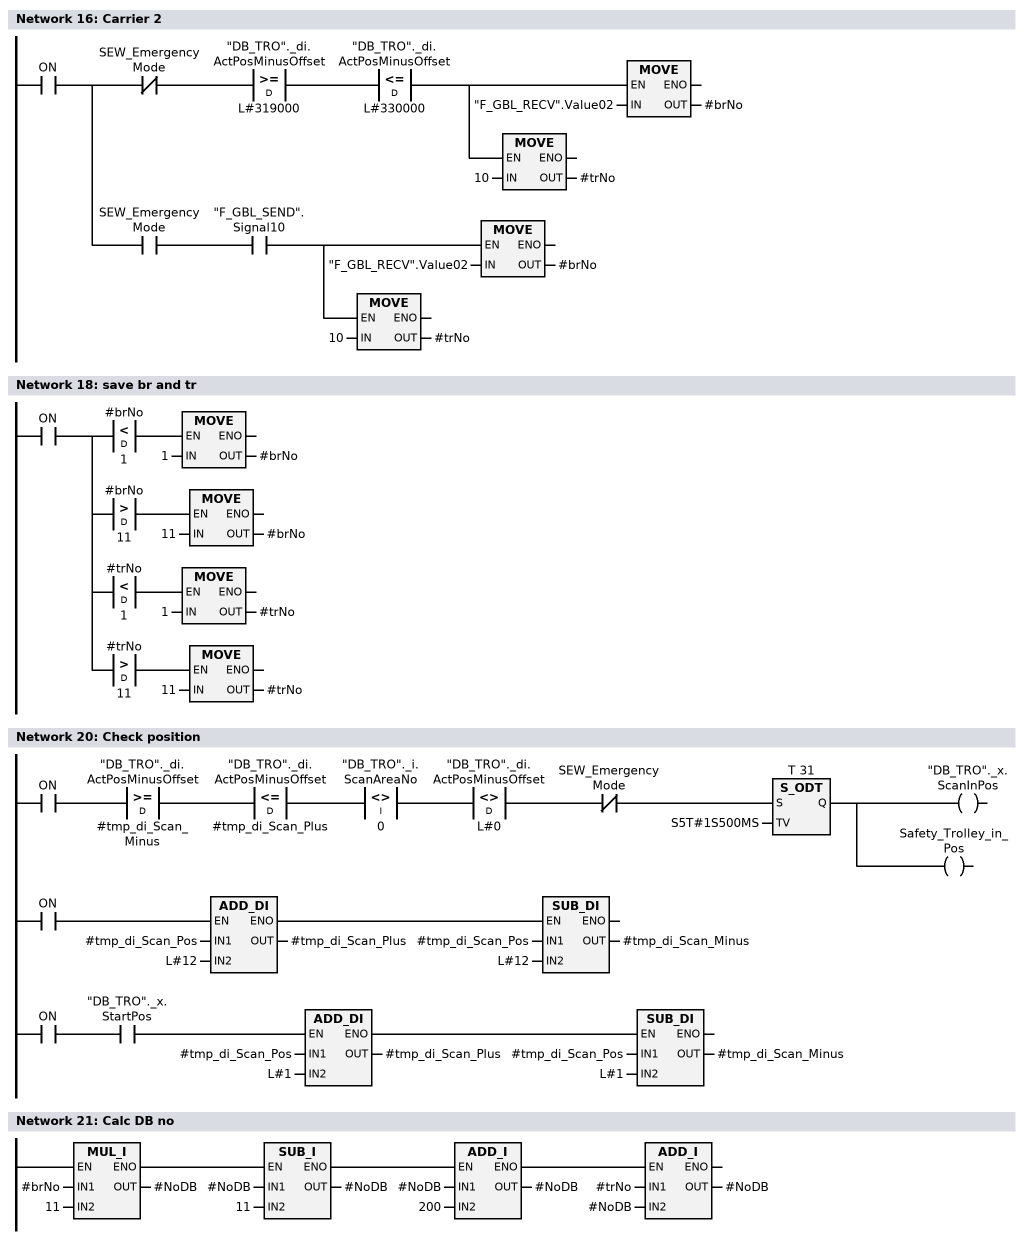
NETWORK
TITLE = Carrier 2
      A     "ON";
      =     L 44.0;
      A     L 44.0;
      AN    "SEW_EmergencyMode";
      A(;
      L     "DB_TRO"._di.ActPosMinusOffset;
      L     L#319000;
      >=D;
      );
      A(;
      L     "DB_TRO"._di.ActPosMinusOffset;
      L     L#330000;
      <=D;
      );
      =     L 44.1;
      A     L 44.1;
      JNB   _01b;
      L     "F_GBL_RECV".Value02;
      T     #brNo;
_01b: NOP   0;
      A     L 44.1;
      JNB   _01c;
      L     10;
      T     #trNo;
_01c: NOP   0;
      A     L 44.0;
      A     "SEW_EmergencyMode";
      A     "F_GBL_SEND".Signal10;
      =     L 44.1;
      A     L 44.1;
      JNB   _01d;
      L     "F_GBL_RECV".Value02;
      T     #brNo;
_01d: NOP   0;
      A     L 44.1;
      JNB   _01e;
      L     10;
      T     #trNo;
_01e: NOP   0;
NETWORK
TITLE = Calc normal row
      L     #trNo;
      L     L#0;
      <>D;
      JC    end;
      L     #startValue;
      L     L#0;
      ==D;
      JC    end;
// we have a row
      L     #brNo;
      L     L#5;
      >D;
      JC    neu;
// old
      L     #startValue;
      L     L#0;	// anpassen auf Achse
      -D;
      DTR;
      L     3.125000e+03;
      /R;
      RND-;
      L     L#2;
      +D;
      T     #trNo;
      JU    end;
// neu
neu:  L     #startValue;
      L     L#0;	// anpassen auf Achse
      -D;
      DTR;
      L     3.500000e+03;
      /R;
      RND-;
      L     L#2;
      +D;
      T     #trNo;
// end
end:  NOP   0;
NETWORK
TITLE = save br and tr
      A     "ON";
      =     L 44.0;
      A     L 44.0;
      A(;
      L     #brNo;
      L     1;
      <D;
      );
      JNB   _01f;
      L     1;
      T     #brNo;
_01f: NOP   0;
      A     L 44.0;
      A(;
      L     #brNo;
      L     11;
      >D;
      );
      JNB   _020;
      L     11;
      T     #brNo;
_020: NOP   0;
      A     L 44.0;
      A(;
      L     #trNo;
      L     1;
      <D;
      );
      JNB   _021;
      L     1;
      T     #trNo;
_021: NOP   0;
      A     L 44.0;
      A(;
      L     #trNo;
      L     11;
      >D;
      );
      JNB   _022;
      L     11;
      T     #trNo;
_022: NOP   0;
NETWORK
TITLE = Get Position
      L     L#0;
      L     "DB_TRO"._i.ScanAreaNo;
      L     1;
      -I;
      L     4;
      *I;
      T     #pMem;
      L     #brNo;
      L     1;
      -I;
      L     44;
      *I;
      L     #pMem;
      +I;
      T     #pMem;
      SLD   3;
      LAR1;
      OPN   "TRO_Positions";
      L     DBD [AR1,P#0.0];
      T     #tmp_di_Scan_Pos;
NETWORK
TITLE = Check position
      A     "ON";
      =     L 44.0;
      A(;
      A     L 44.0;
      JNB   _023;
      L     #tmp_di_Scan_Pos;
      L     L#12;
      +D;
      T     #tmp_di_Scan_Plus;
      AN    OV;
      SAVE;
      CLR;
_023: A     BR;
      );
      JNB   _024;
      L     #tmp_di_Scan_Pos;
      L     L#12;
      -D;
      T     #tmp_di_Scan_Minus;
_024: NOP   0;
      A(;
      A     L 44.0;
      A     "DB_TRO"._x.StartPos;
      JNB   _025;
      L     #tmp_di_Scan_Pos;
      L     L#1;
      +D;
      T     #tmp_di_Scan_Plus;
      AN    OV;
      SAVE;
      CLR;
_025: A     BR;
      );
      JNB   _026;
      L     #tmp_di_Scan_Pos;
      L     L#1;
      -D;
      T     #tmp_di_Scan_Minus;
_026: NOP   0;
      A     L 44.0;
      A(;
      L     "DB_TRO"._di.ActPosMinusOffset;
      L     #tmp_di_Scan_Minus;
      >=D;
      );
      A(;
      L     "DB_TRO"._di.ActPosMinusOffset;
      L     #tmp_di_Scan_Plus;
      <=D;
      );
      A(;
      L     "DB_TRO"._i.ScanAreaNo;
      L     0;
      <>I;
      );
      A(;
      L     "DB_TRO"._di.ActPosMinusOffset;
      L     L#0;
      <>D;
      );
      AN    "SEW_EmergencyMode";
      L     S5T#1S500MS;
      SD    T 31;
      NOP   0;
      NOP   0;
      NOP   0;
      A     T 31;
      =     "DB_TRO"._x.ScanInPos;
      =     "Safety_Trolley_in_Pos";
NETWORK
TITLE = Calc DB no
      A(;
      A(;
      A(;
      L     #brNo;
      L     11;
      *I;
      T     #NoDB;
      AN    OV;
      SAVE;
      CLR;
      A     BR;
      );
      JNB   _027;
      L     #NoDB;
      L     11;
      -I;
      T     #NoDB;
      AN    OV;
      SAVE;
      CLR;
_027: A     BR;
      );
      JNB   _028;
      L     #NoDB;
      L     200;
      +I;
      T     #NoDB;
      AN    OV;
      SAVE;
      CLR;
_028: A     BR;
      );
      JNB   _029;
      L     #trNo;
      L     #NoDB;
      +I;
      T     #NoDB;
_029: NOP   0;
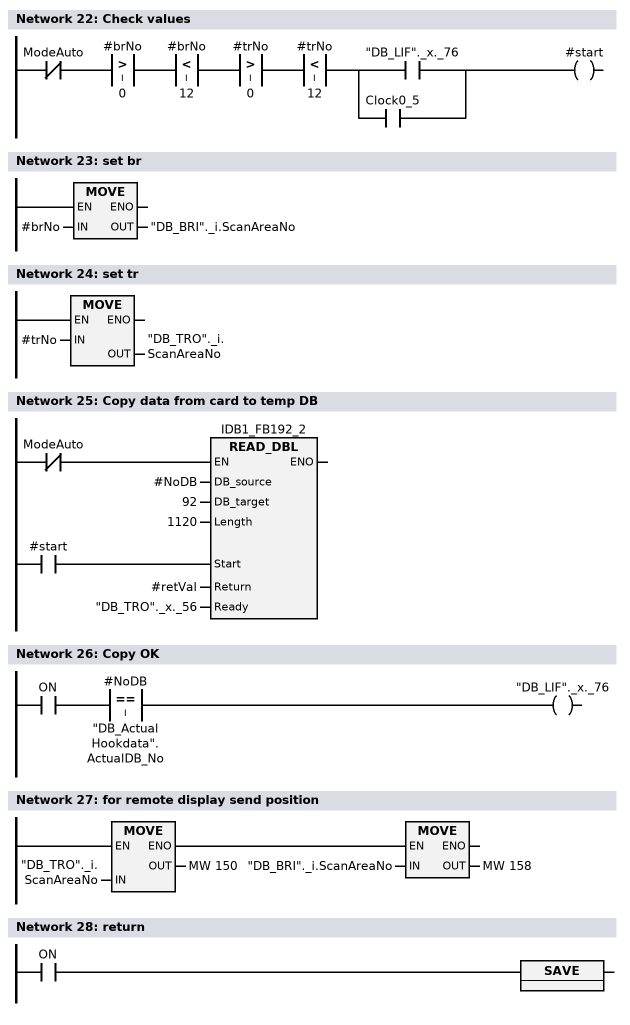
NETWORK
TITLE = Check values
      AN    "ModeAuto";
      A(;
      L     #brNo;
      L     0;
      >I;
      );
      A(;
      L     #brNo;
      L     12;
      <I;
      );
      A(;
      L     #trNo;
      L     0;
      >I;
      );
      A(;
      L     #trNo;
      L     12;
      <I;
      );
      A(;
      O     "DB_LIF"._x._76;
      O     "Clock0_5";
      );
      =     #start;
NETWORK
TITLE = set br
      L     #brNo;
      T     "DB_BRI"._i.ScanAreaNo;
      NOP   0;
NETWORK
TITLE = set tr
      L     #trNo;
      T     "DB_TRO"._i.ScanAreaNo;
      NOP   0;
NETWORK
TITLE = Copy data from card to temp DB
      A     #start;
      =     L 44.0;
      BLD   103;
      AN    "ModeAuto";
      JNB   _02a;
      CALL  "READ_DBL" , "IDB1_FB192_2" (
           DB_source                := #NoDB,
           DB_target                := 92,
           Length                   := 1120,
           Start                    := L 44.0,
           Return                   := #retVal,
           Ready                    := "DB_TRO"._x._56);
_02a: NOP   0;
NETWORK
TITLE = Copy OK
      A     "ON";
      A(;
      L     #NoDB;
      L     "DB_ActualHookdata".ActualDB_No;
      ==I;
      );
      =     "DB_LIF"._x._76;
NETWORK
TITLE = for remote display send position
      A(;
      L     "DB_TRO"._i.ScanAreaNo;
      T     MW 150;
      SET;
      SAVE;
      CLR;
      A     BR;
      );
      JNB   _02b;
      L     "DB_BRI"._i.ScanAreaNo;
      T     MW 158;
_02b: NOP   0;
NETWORK
TITLE = return
      A     "ON";
      SAVE;
END_FUNCTION

FUNCTION "Axis_TROLLEY_Scan_Man" : VOID	// FC 215
TITLE = Scan manual pos
//
//Baustein-Kommentar ...
//
AUTHOR : Koenig
FAMILY : Scan
NAME : ManPos
VERSION : 1.0
VAR_INPUT
  BridgeNo : INT ;	//Bridge position no
  PositionNo : INT ;	//Positions number
  PositionDB : INT ;	//DB Number of Positions
  ActualPosition : DINT ;
  PositionMin : DINT ;
  PositionMax : DINT ;
END_VAR
VAR_OUTPUT
  PrevPosition : DINT ;
  NextPosition : DINT ;
  FirstPosition : DINT ;
  LastPosition : DINT ;
  Error : WORD ;
END_VAR
VAR_TEMP
  i : INT ;
  value : DINT ;
  diff : DINT ;
  DB_No : WORD ;
  DB_Length : WORD ;
  DB_WP : BOOL ;
  RETURN_Value : INT ;
END_VAR
BEGIN
// body was compiled from an SCL source; compiled code not shown
END_FUNCTION

FUNCTION "Axis_TROLLEY_Flt_065-080" : VOID	// FC 219
TITLE = Error Trolley 65-80
VERSION : 0.1
BEGIN
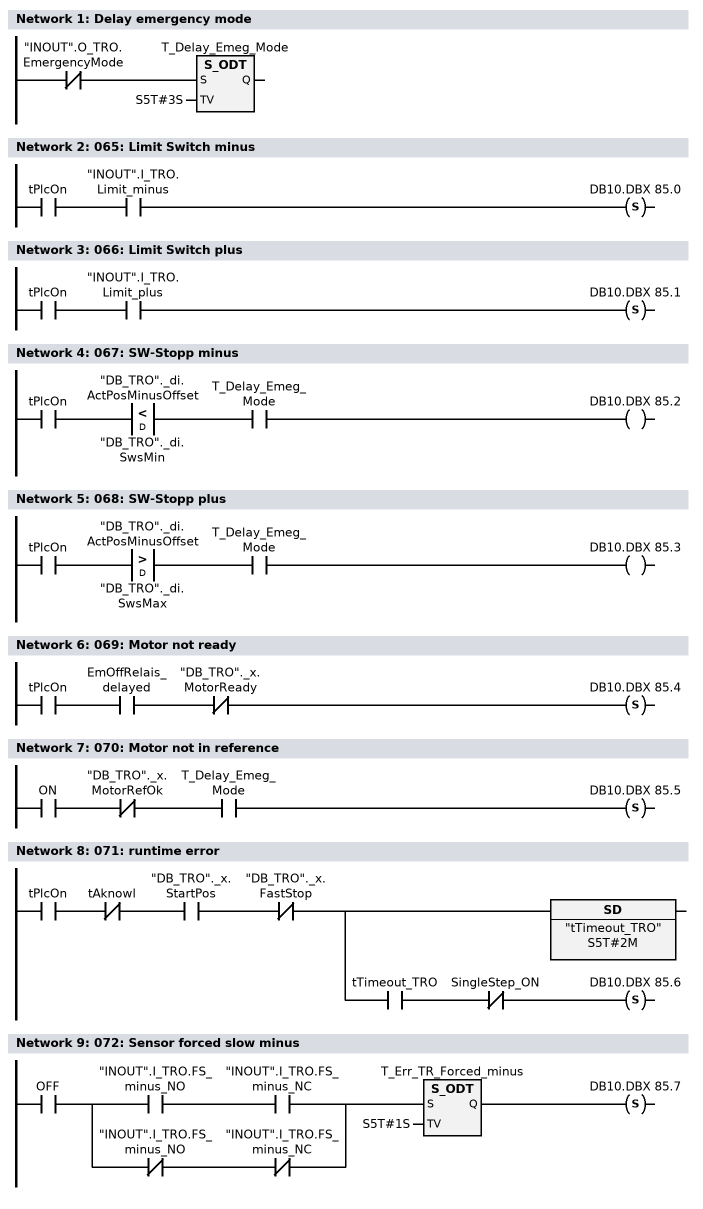
NETWORK
TITLE = Delay emergency mode
      AN    "INOUT".O_TRO.EmergencyMode;
      L     S5T#3S;
      SD    "T_Delay_Emeg_Mode";
      NOP   0;
      NOP   0;
      NOP   0;
      NOP   0;
NETWORK
TITLE = 065: Limit Switch minus
      A     "tPlcOn";
      A     "INOUT".I_TRO.Limit_minus;
      S     DB10.DBX 85.0;
NETWORK
TITLE = 066: Limit Switch plus
      A     "tPlcOn";
      A     "INOUT".I_TRO.Limit_plus;
      S     DB10.DBX 85.1;
NETWORK
TITLE = 067: SW-Stopp minus
      A     "tPlcOn";
      A(;
      L     "DB_TRO"._di.ActPosMinusOffset;
      L     "DB_TRO"._di.SwsMin;
      <D;
      );
      A     "T_Delay_Emeg_Mode";
      =     DB10.DBX 85.2;
NETWORK
TITLE = 068: SW-Stopp plus
      A     "tPlcOn";
      A(;
      L     "DB_TRO"._di.ActPosMinusOffset;
      L     "DB_TRO"._di.SwsMax;
      >D;
      );
      A     "T_Delay_Emeg_Mode";
      =     DB10.DBX 85.3;
NETWORK
TITLE = 069: Motor not ready
      A     "tPlcOn";
      A     "EmOffRelais_delayed";
      AN    "DB_TRO"._x.MotorReady;
      S     DB10.DBX 85.4;
NETWORK
TITLE = 070: Motor not in reference
      A     "ON";
      AN    "DB_TRO"._x.MotorRefOk;
      A     "T_Delay_Emeg_Mode";
      S     DB10.DBX 85.5;
NETWORK
TITLE = 071: runtime error
      A     "tPlcOn";
      AN    "tAknowl";
      A     "DB_TRO"._x.StartPos;
      AN    "DB_TRO"._x.FastStop;
      =     L 0.0;
      A     L 0.0;
      BLD   102;
      L     S5T#2M;
      SD    "tTimeout_TRO";
      A     L 0.0;
      A     "tTimeout_TRO";
      AN    "SingleStep_ON";
      S     DB10.DBX 85.6;
NETWORK
TITLE = 072: Sensor forced slow minus
      A     "OFF";
      A(;
      A     "INOUT".I_TRO.FS_minus_NO;
      A     "INOUT".I_TRO.FS_minus_NC;
      O;
      AN    "INOUT".I_TRO.FS_minus_NO;
      AN    "INOUT".I_TRO.FS_minus_NC;
      );
      L     S5T#1S;
      SD    "T_Err_TR_Forced_minus";
      NOP   0;
      NOP   0;
      NOP   0;
      A     "T_Err_TR_Forced_minus";
      S     DB10.DBX 85.7;
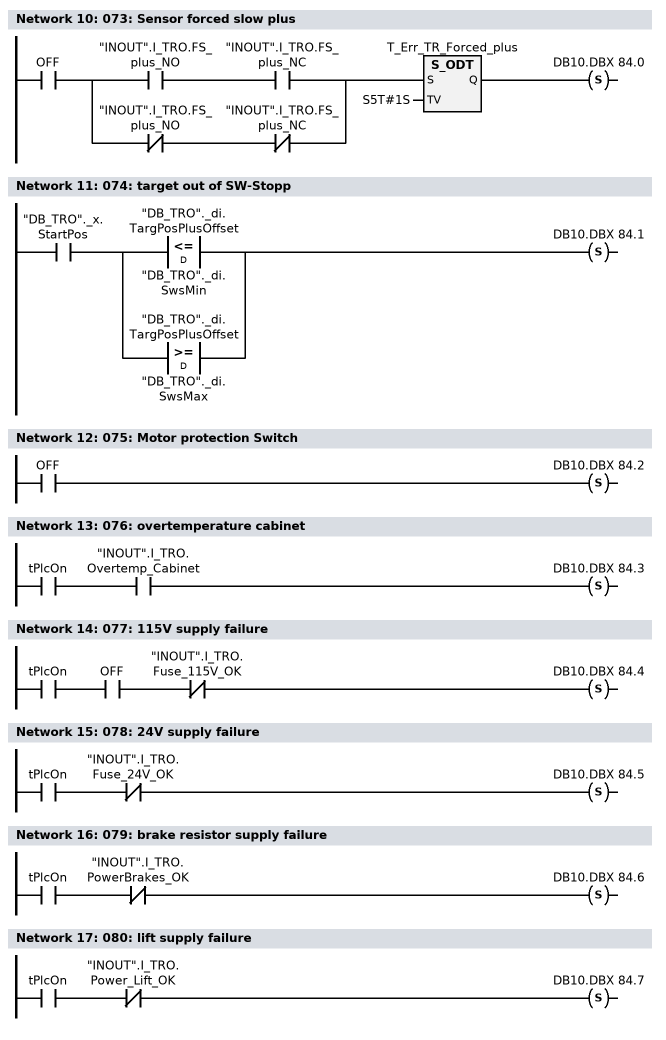
NETWORK
TITLE = 073: Sensor forced slow plus
      A     "OFF";
      A(;
      A     "INOUT".I_TRO.FS_plus_NO;
      A     "INOUT".I_TRO.FS_plus_NC;
      O;
      AN    "INOUT".I_TRO.FS_plus_NO;
      AN    "INOUT".I_TRO.FS_plus_NC;
      );
      L     S5T#1S;
      SD    "T_Err_TR_Forced_plus";
      NOP   0;
      NOP   0;
      NOP   0;
      A     "T_Err_TR_Forced_plus";
      S     DB10.DBX 84.0;
NETWORK
TITLE = 074: target out of SW-Stopp
      A     "DB_TRO"._x.StartPos;
      A(;
      O(;
      L     "DB_TRO"._di.TargPosPlusOffset;
      L     "DB_TRO"._di.SwsMin;
      <=D;
      );
      O(;
      L     "DB_TRO"._di.TargPosPlusOffset;
      L     "DB_TRO"._di.SwsMax;
      >=D;
      );
      );
      S     DB10.DBX 84.1;
NETWORK
TITLE = 075: Motor protection Switch
      A     "OFF";
      S     DB10.DBX 84.2;
NETWORK
TITLE = 076: overtemperature cabinet
      A     "tPlcOn";
      A     "INOUT".I_TRO.Overtemp_Cabinet;
      S     DB10.DBX 84.3;
NETWORK
TITLE = 077: 115V supply failure
      A     "tPlcOn";
      A     "OFF";
      AN    "INOUT".I_TRO.Fuse_115V_OK;
      S     DB10.DBX 84.4;
NETWORK
TITLE = 078: 24V supply failure
      A     "tPlcOn";
      AN    "INOUT".I_TRO.Fuse_24V_OK;
      S     DB10.DBX 84.5;
NETWORK
TITLE = 079: brake resistor supply failure
//14 
      A     "tPlcOn";
      AN    "INOUT".I_TRO.PowerBrakes_OK;
      S     DB10.DBX 84.6;
NETWORK
TITLE = 080: lift supply failure
      A     "tPlcOn";
      AN    "INOUT".I_TRO.Power_Lift_OK;
      S     DB10.DBX 84.7;
END_FUNCTION

FUNCTION "Axis_LIFT" : VOID	// FC 220
TITLE = Axis LIFT
VERSION : 0.1
VAR_TEMP
  tmp_RetVal : INT ;
  tmp_RetVal2 : INT ;
  tmp_SourceDB1 : INT ;
  tmp_SourceDB2 : INT ;
  tmp_TargetDB1 : INT ;
  tmp_TargetDB2 : INT ;
  tmp_StartDBCopy : BOOL ;
  tmp_ReadDB_OK : BOOL ;
END_VAR
BEGIN
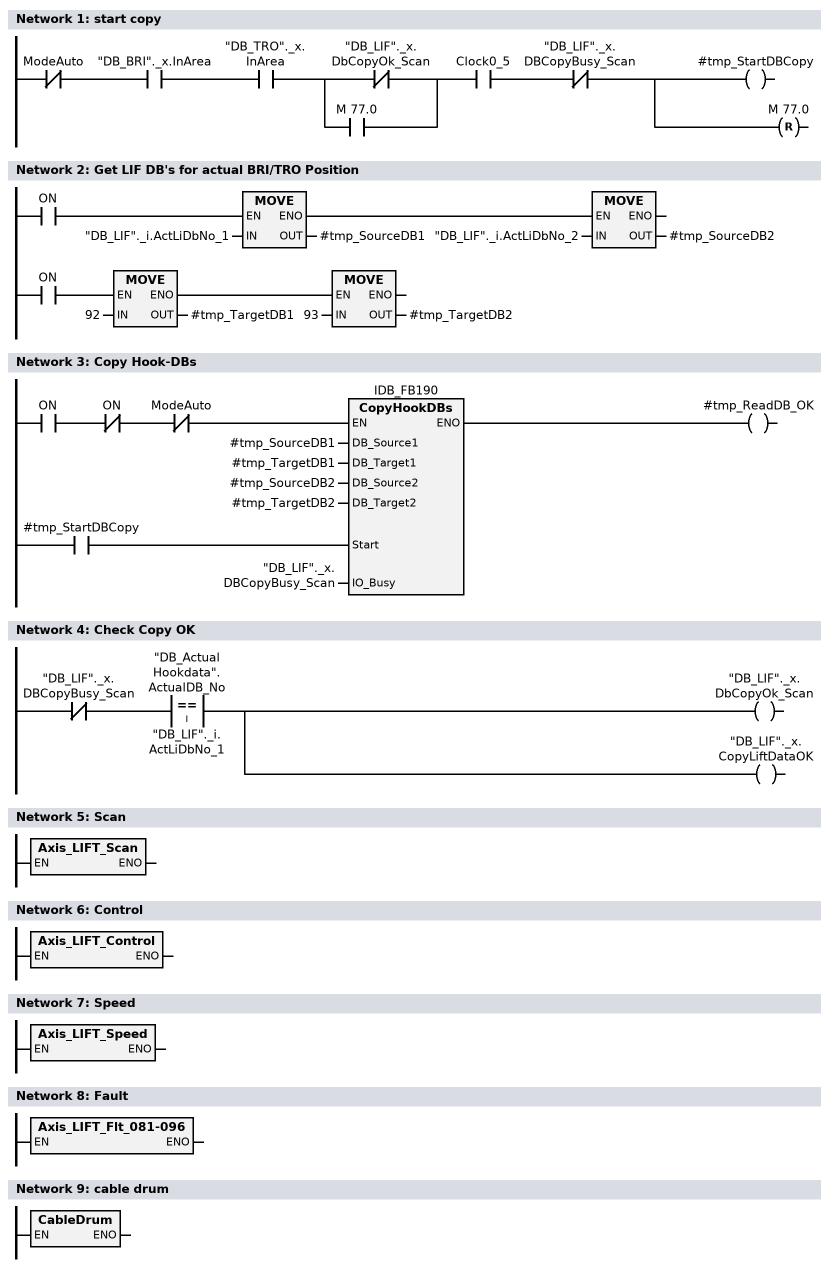
NETWORK
TITLE = start copy
      AN    "ModeAuto";
      A     "DB_BRI"._x.InArea;
      A     "DB_TRO"._x.InArea;
      A(;
      ON    "DB_LIF"._x.DbCopyOk_Scan;
      O     M 77.0;
      );
      A     "Clock0_5";
      AN    "DB_LIF"._x.DBCopyBusy_Scan;
      =     #tmp_StartDBCopy;
      R     M 77.0;
NETWORK
TITLE = Get LIF DB's for actual BRI/TRO Position
//Actual DB from Scan BRI
//
      A     "ON";
      =     L 13.0;
      A(;
      A     L 13.0;
      JNB   _001;
      L     "DB_LIF"._i.ActLiDbNo_1;
      T     #tmp_SourceDB1;
      SET;
      SAVE;
      CLR;
_001: A     BR;
      );
      JNB   _002;
      L     "DB_LIF"._i.ActLiDbNo_2;
      T     #tmp_SourceDB2;
_002: NOP   0;
      A(;
      A     L 13.0;
      JNB   _003;
      L     92;
      T     #tmp_TargetDB1;
      SET;
      SAVE;
      CLR;
_003: A     BR;
      );
      JNB   _004;
      L     93;
      T     #tmp_TargetDB2;
_004: NOP   0;
NETWORK
TITLE = Copy Hook-DBs
      A     #tmp_StartDBCopy;
      =     L 13.0;
      BLD   103;
      A     "ON";
      AN    "ON";
      AN    "ModeAuto";
      JNB   _005;
      CALL  "CopyHookDBs" , "IDB_FB190" (
           DB_Source1               := #tmp_SourceDB1,
           DB_Target1               := #tmp_TargetDB1,
           DB_Source2               := #tmp_SourceDB2,
           DB_Target2               := #tmp_TargetDB2,
           Start                    := L 13.0,
           IO_Busy                  := "DB_LIF"._x.DBCopyBusy_Scan);
_005: A     BR;
      =     #tmp_ReadDB_OK;
NETWORK
TITLE = Check Copy OK
      AN    "DB_LIF"._x.DBCopyBusy_Scan;
      A(;
      L     "DB_ActualHookdata".ActualDB_No;
      L     "DB_LIF"._i.ActLiDbNo_1;
      ==I;
      );
      =     "DB_LIF"._x.DbCopyOk_Scan;
      =     "DB_LIF"._x.CopyLiftDataOK;
NETWORK
TITLE = Scan
      CALL  "Axis_LIFT_Scan";
      NOP   0;
NETWORK
TITLE = Control
      CALL  "Axis_LIFT_Control";
      NOP   0;
NETWORK
TITLE = Speed
      CALL  "Axis_LIFT_Speed";
      NOP   0;
NETWORK
TITLE = Fault
      CALL  "Axis_LIFT_Flt_081-096";
      NOP   0;
NETWORK
TITLE = cable drum
      CALL  "CableDrum";
      NOP   0;
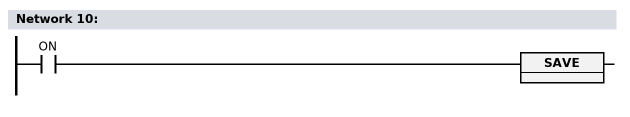
NETWORK
TITLE =
      A     "ON";
      SAVE;
END_FUNCTION

FUNCTION "Axis_LIFT_Control" : VOID	// FC 222
TITLE = LIFT Control
VERSION : 0.1
VAR_TEMP
  tmp_Targ_HO_1_auto : BOOL ;
  tmp_Targ_HO_2_auto : BOOL ;
  tmp_Targ_HO_3_auto : BOOL ;
  tmp_Targ_HO_1_man : BOOL ;
  tmp_Targ_HU_1_auto : BOOL ;
  tmp_Targ_HU_2_auto : BOOL ;
  tmp_Targ_HU_1_man : BOOL ;
  tmp_Targ_Intern_1_auto : BOOL ;
  tmp_Targ_Intern_2_auto : BOOL ;
  tmp_Targ_Intern_3_auto : BOOL ;
  tmp_Targ_Top_auto : BOOL ;
  tmp_Targ_Top_man : BOOL ;
  tmp_switch : BOOL ;
  TargetOK : BOOL ;
  TargetValueOK : BOOL ;
  tmp_InPos : BOOL ;
  tmp_Rel_MaxDis : BOOL ;
  modePos : BOOL ;
  modeInch : BOOL ;
  tmp_Targ_Man : BOOL ;
  tmp_DIR : BOOL ;
  tmp_di_DiffPos : DINT ;
  prev : DINT ;
  next : DINT ;
  min : DINT ;
  max : DINT ;
END_VAR
BEGIN
NETWORK
TITLE =
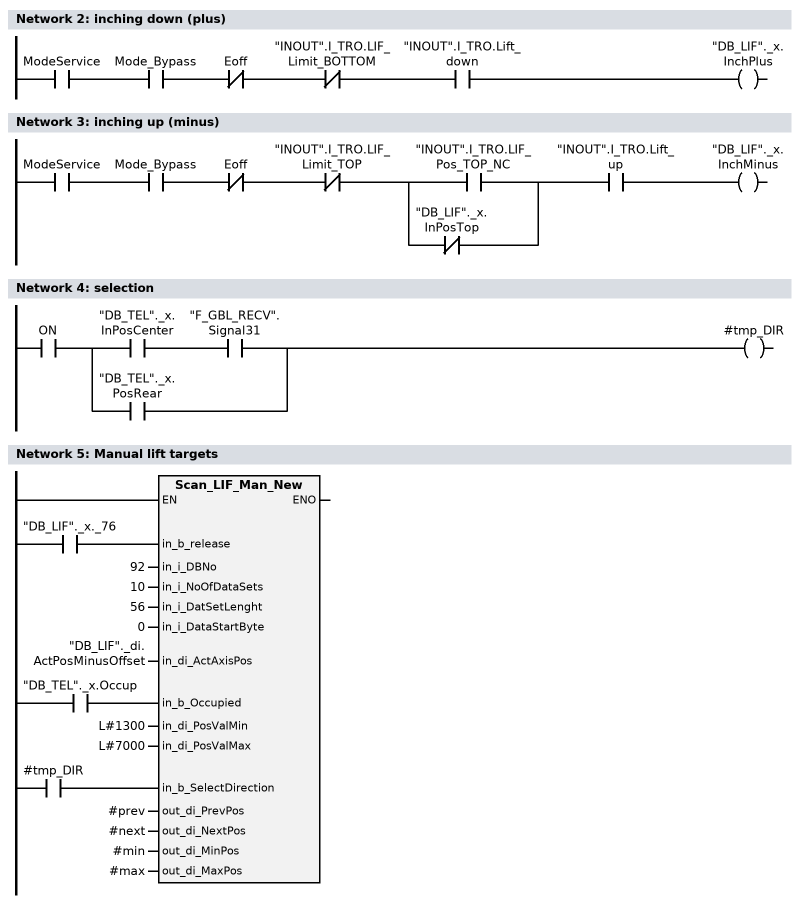
NETWORK
TITLE = inching down (plus)
      A     "ModeService";
      A     "Mode_Bypass";
      AN    "Eoff";
      AN    "INOUT".I_TRO.LIF_Limit_BOTTOM;
      A     "INOUT".I_TRO.Lift_down;
      =     "DB_LIF"._x.InchPlus;
NETWORK
TITLE = inching up (minus)
      A     "ModeService";
      A     "Mode_Bypass";
      AN    "Eoff";
      AN    "INOUT".I_TRO.LIF_Limit_TOP;
      A(;
      O     "INOUT".I_TRO.LIF_Pos_TOP_NC;
      ON    "DB_LIF"._x.InPosTop;
      );
      A     "INOUT".I_TRO.Lift_up;
      =     "DB_LIF"._x.InchMinus;
NETWORK
TITLE = selection
      A     "ON";
      A(;
      A     "DB_TEL"._x.InPosCenter;
      A     "F_GBL_RECV".Signal31;
      O     "DB_TEL"._x.PosRear;
      );
      =     #tmp_DIR;
NETWORK
TITLE = Manual lift targets
      A     "DB_LIF"._x._76;
      =     L 24.0;
      BLD   103;
      A     "DB_TEL"._x.Occup;
      =     L 24.1;
      BLD   103;
      A     #tmp_DIR;
      =     L 24.2;
      BLD   103;
      CALL  "Scan_LIF_Man_New" (
           in_b_release             := L 24.0,
           in_i_DBNo                := 92,
           in_i_NoOfDataSets        := 10,
           in_i_DatSetLenght        := 56,
           in_i_DataStartByte       := 0,
           in_di_ActAxisPos         := "DB_LIF"._di.ActPosMinusOffset,
           in_b_Occupied            := L 24.1,
           in_di_PosValMin          := L#1300,
           in_di_PosValMax          := L#7000,
           in_b_SelectDirection     := L 24.2,
           out_di_PrevPos           := #prev,
           out_di_NextPos           := #next,
           out_di_MinPos            := #min,
           out_di_MaxPos            := #max);
      NOP   0;
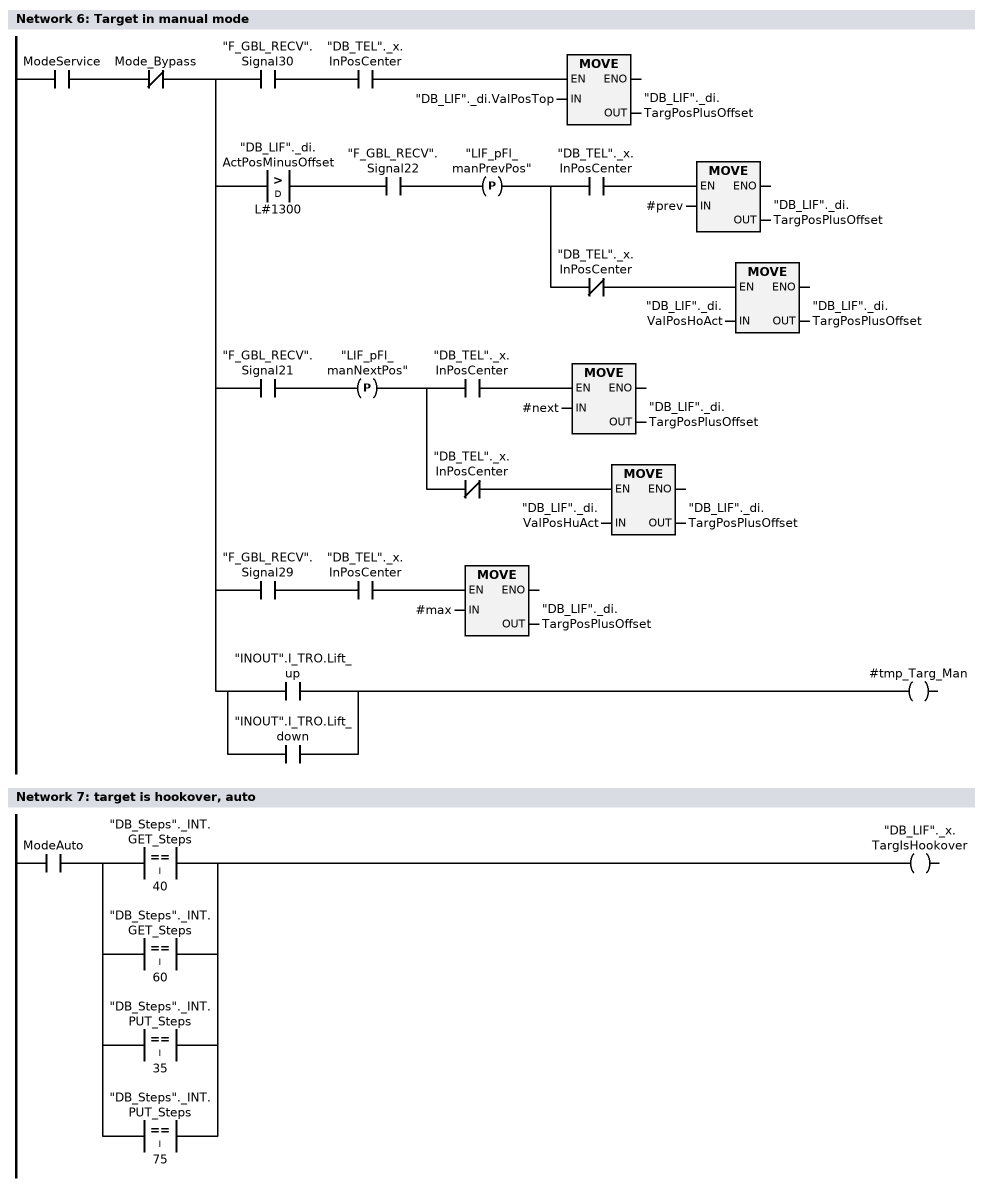
NETWORK
TITLE = Target in manual mode
      A     "ModeService";
      AN    "Mode_Bypass";
      =     L 24.0;
      A     L 24.0;
      A     "F_GBL_RECV".Signal30;
      A     "DB_TEL"._x.InPosCenter;
      JNB   _001;
      L     "DB_LIF"._di.ValPosTop;
      T     "DB_LIF"._di.TargPosPlusOffset;
_001: NOP   0;
      A     L 24.0;
      A(;
      L     "DB_LIF"._di.ActPosMinusOffset;
      L     L#1300;
      >D;
      );
      A     "F_GBL_RECV".Signal22;
      FP    "LIF_pFl_manPrevPos";
      =     L 24.1;
      A     L 24.1;
      A     "DB_TEL"._x.InPosCenter;
      JNB   _002;
      L     #prev;
      T     "DB_LIF"._di.TargPosPlusOffset;
_002: NOP   0;
      A     L 24.1;
      AN    "DB_TEL"._x.InPosCenter;
      JNB   _003;
      L     "DB_LIF"._di.ValPosHoAct;
      T     "DB_LIF"._di.TargPosPlusOffset;
_003: NOP   0;
      A     L 24.0;
      A     "F_GBL_RECV".Signal21;
      FP    "LIF_pFl_manNextPos";
      =     L 24.1;
      A     L 24.1;
      A     "DB_TEL"._x.InPosCenter;
      JNB   _004;
      L     #next;
      T     "DB_LIF"._di.TargPosPlusOffset;
_004: NOP   0;
      A     L 24.1;
      AN    "DB_TEL"._x.InPosCenter;
      JNB   _005;
      L     "DB_LIF"._di.ValPosHuAct;
      T     "DB_LIF"._di.TargPosPlusOffset;
_005: NOP   0;
      A     L 24.0;
      A     "F_GBL_RECV".Signal29;
      A     "DB_TEL"._x.InPosCenter;
      JNB   _006;
      L     #max;
      T     "DB_LIF"._di.TargPosPlusOffset;
_006: NOP   0;
      A     L 24.0;
      A(;
      O     "INOUT".I_TRO.Lift_up;
      O     "INOUT".I_TRO.Lift_down;
      );
      =     #tmp_Targ_Man;
NETWORK
TITLE = target is hookover, auto
      A     "ModeAuto";
      A(;
      O(;
      L     "DB_Steps"._INT.GET_Steps;
      L     40;
      ==I;
      );
      O(;
      L     "DB_Steps"._INT.GET_Steps;
      L     60;
      ==I;
      );
      O(;
      L     "DB_Steps"._INT.PUT_Steps;
      L     35;
      ==I;
      );
      O(;
      L     "DB_Steps"._INT.PUT_Steps;
      L     75;
      ==I;
      );
      );
      =     "DB_LIF"._x.TargIsHookover;
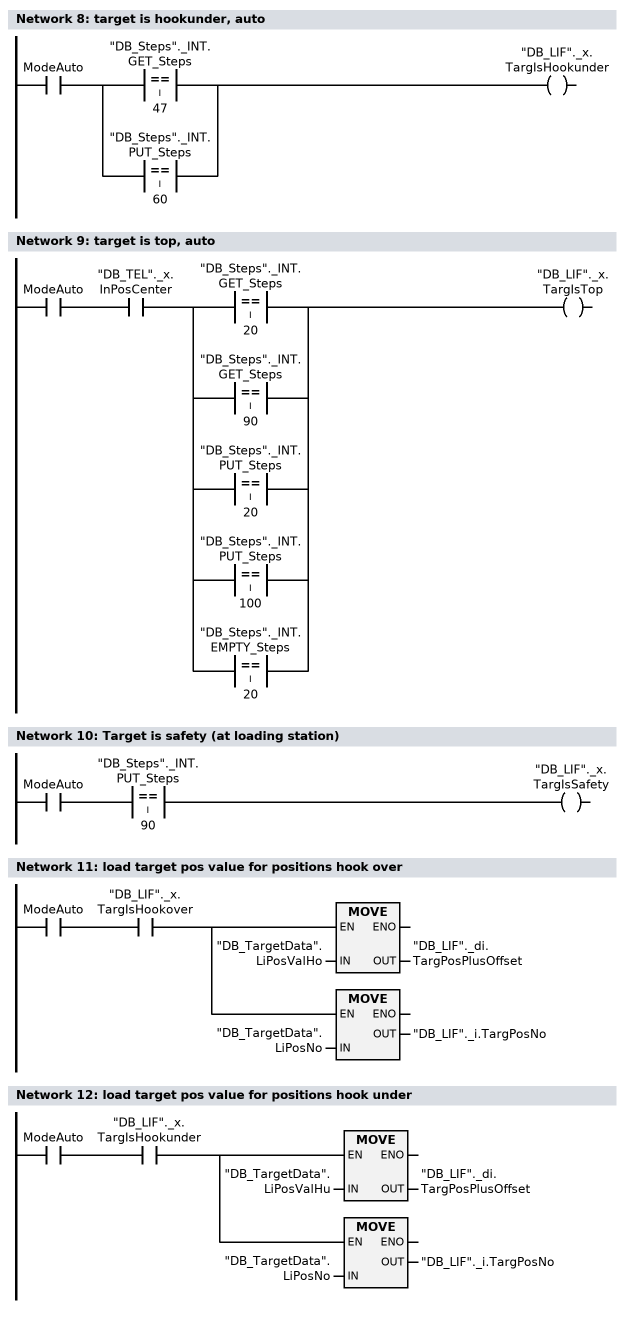
NETWORK
TITLE = target is hookunder, auto
      A     "ModeAuto";
      A(;
      O(;
      L     "DB_Steps"._INT.GET_Steps;
      L     47;
      ==I;
      );
      O(;
      L     "DB_Steps"._INT.PUT_Steps;
      L     60;
      ==I;
      );
      );
      =     "DB_LIF"._x.TargIsHookunder;
NETWORK
TITLE = target is top, auto
      A     "ModeAuto";
      A     "DB_TEL"._x.InPosCenter;
      A(;
      O(;
      L     "DB_Steps"._INT.GET_Steps;
      L     20;
      ==I;
      );
      O(;
      L     "DB_Steps"._INT.GET_Steps;
      L     90;
      ==I;
      );
      O(;
      L     "DB_Steps"._INT.PUT_Steps;
      L     20;
      ==I;
      );
      O(;
      L     "DB_Steps"._INT.PUT_Steps;
      L     100;
      ==I;
      );
      O(;
      L     "DB_Steps"._INT.EMPTY_Steps;
      L     20;
      ==I;
      );
      );
      =     "DB_LIF"._x.TargIsTop;
NETWORK
TITLE = Target is safety (at loading station)
      A     "ModeAuto";
      A(;
      L     "DB_Steps"._INT.PUT_Steps;
      L     90;
      ==I;
      );
      =     "DB_LIF"._x.TargIsSafety;
NETWORK
TITLE = load target pos value for positions hook over
      A     "ModeAuto";
      A     "DB_LIF"._x.TargIsHookover;
      =     L 24.0;
      A     L 24.0;
      JNB   _007;
      L     "DB_TargetData".LiPosValHo;
      T     "DB_LIF"._di.TargPosPlusOffset;
_007: NOP   0;
      A     L 24.0;
      JNB   _008;
      L     "DB_TargetData".LiPosNo;
      T     "DB_LIF"._i.TargPosNo;
_008: NOP   0;
NETWORK
TITLE = load target pos value for positions hook under
      A     "ModeAuto";
      A     "DB_LIF"._x.TargIsHookunder;
      =     L 24.0;
      A     L 24.0;
      JNB   _009;
      L     "DB_TargetData".LiPosValHu;
      T     "DB_LIF"._di.TargPosPlusOffset;
_009: NOP   0;
      A     L 24.0;
      JNB   _00a;
      L     "DB_TargetData".LiPosNo;
      T     "DB_LIF"._i.TargPosNo;
_00a: NOP   0;
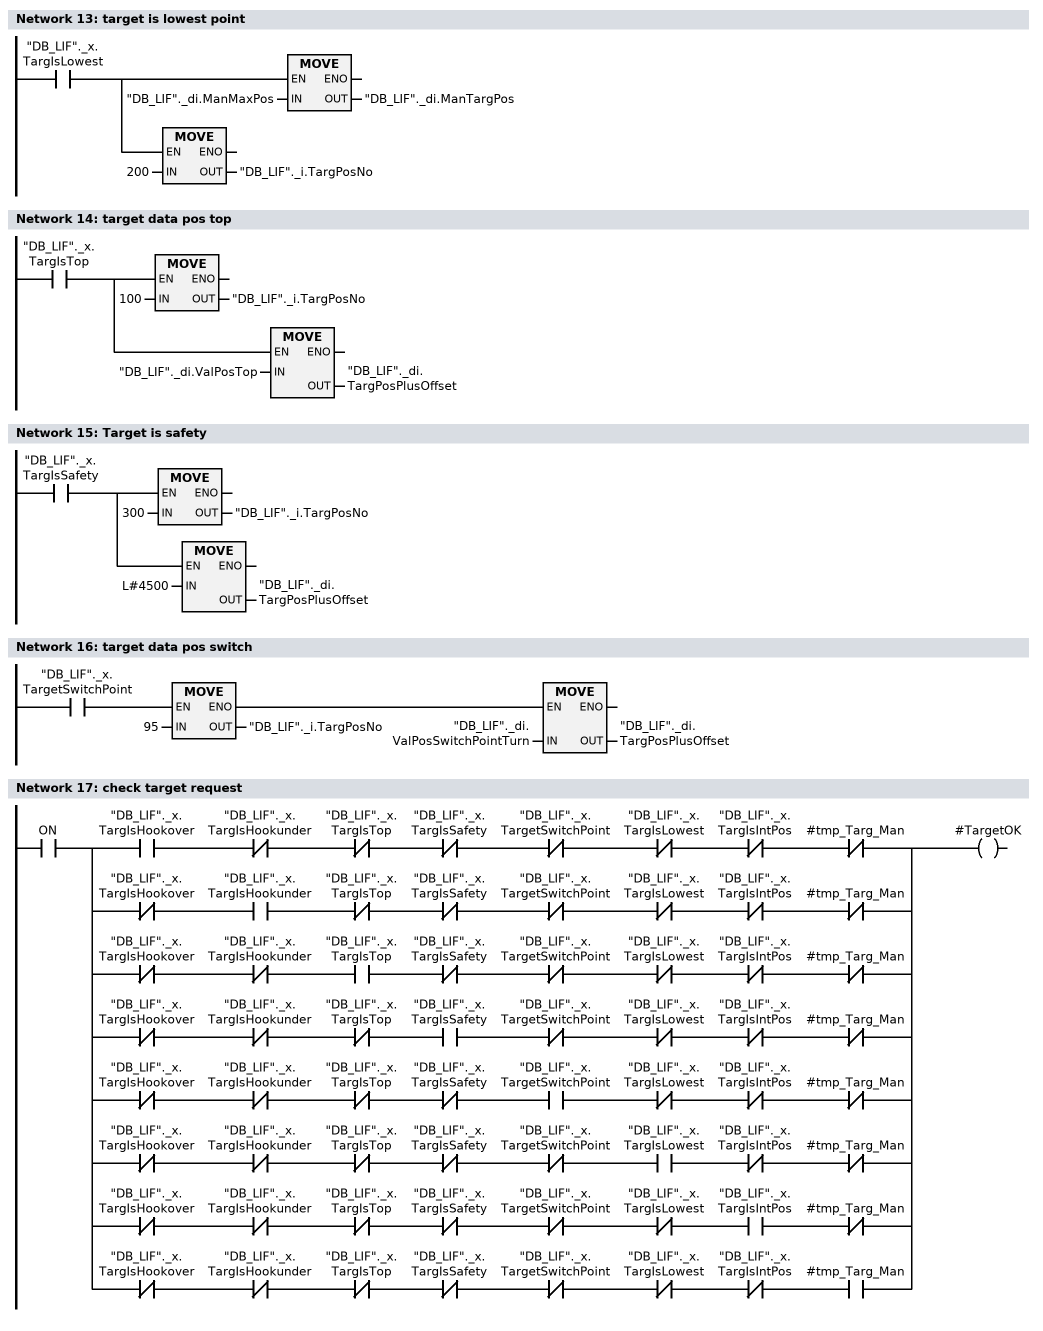
NETWORK
TITLE = target is lowest point
      A     "DB_LIF"._x.TargIsLowest;
      =     L 24.0;
      A     L 24.0;
      JNB   _00b;
      L     "DB_LIF"._di.ManMaxPos;
      T     "DB_LIF"._di.ManTargPos;
_00b: NOP   0;
      A     L 24.0;
      JNB   _00c;
      L     200;
      T     "DB_LIF"._i.TargPosNo;
_00c: NOP   0;
NETWORK
TITLE = target data pos top
      A     "DB_LIF"._x.TargIsTop;
      =     L 24.0;
      A     L 24.0;
      JNB   _00d;
      L     100;
      T     "DB_LIF"._i.TargPosNo;
_00d: NOP   0;
      A     L 24.0;
      JNB   _00e;
      L     "DB_LIF"._di.ValPosTop;
      T     "DB_LIF"._di.TargPosPlusOffset;
_00e: NOP   0;
NETWORK
TITLE = Target is safety
      A     "DB_LIF"._x.TargIsSafety;
      =     L 24.0;
      A     L 24.0;
      JNB   _00f;
      L     300;
      T     "DB_LIF"._i.TargPosNo;
_00f: NOP   0;
      A     L 24.0;
      JNB   _010;
      L     L#4500;
      T     "DB_LIF"._di.TargPosPlusOffset;
_010: NOP   0;
NETWORK
TITLE = target data pos switch
      A(;
      A     "DB_LIF"._x.TargetSwitchPoint;
      JNB   _011;
      L     95;
      T     "DB_LIF"._i.TargPosNo;
      SET;
      SAVE;
      CLR;
_011: A     BR;
      );
      JNB   _012;
      L     "DB_LIF"._di.ValPosSwitchPointTurn;
      T     "DB_LIF"._di.TargPosPlusOffset;
_012: NOP   0;
NETWORK
TITLE = check target request
//only allow one target otherwise values are wrong !
      A     "ON";
      A(;
      A     "DB_LIF"._x.TargIsHookover;
      AN    "DB_LIF"._x.TargIsHookunder;
      AN    "DB_LIF"._x.TargIsTop;
      AN    "DB_LIF"._x.TargIsSafety;
      AN    "DB_LIF"._x.TargetSwitchPoint;
      AN    "DB_LIF"._x.TargIsLowest;
      AN    "DB_LIF"._x.TargIsIntPos;
      AN    #tmp_Targ_Man;
      O;
      AN    "DB_LIF"._x.TargIsHookover;
      A     "DB_LIF"._x.TargIsHookunder;
      AN    "DB_LIF"._x.TargIsTop;
      AN    "DB_LIF"._x.TargIsSafety;
      AN    "DB_LIF"._x.TargetSwitchPoint;
      AN    "DB_LIF"._x.TargIsLowest;
      AN    "DB_LIF"._x.TargIsIntPos;
      AN    #tmp_Targ_Man;
      O;
      AN    "DB_LIF"._x.TargIsHookover;
      AN    "DB_LIF"._x.TargIsHookunder;
      A     "DB_LIF"._x.TargIsTop;
      AN    "DB_LIF"._x.TargIsSafety;
      AN    "DB_LIF"._x.TargetSwitchPoint;
      AN    "DB_LIF"._x.TargIsLowest;
      AN    "DB_LIF"._x.TargIsIntPos;
      AN    #tmp_Targ_Man;
      O;
      AN    "DB_LIF"._x.TargIsHookover;
      AN    "DB_LIF"._x.TargIsHookunder;
      AN    "DB_LIF"._x.TargIsTop;
      A     "DB_LIF"._x.TargIsSafety;
      AN    "DB_LIF"._x.TargetSwitchPoint;
      AN    "DB_LIF"._x.TargIsLowest;
      AN    "DB_LIF"._x.TargIsIntPos;
      AN    #tmp_Targ_Man;
      O;
      AN    "DB_LIF"._x.TargIsHookover;
      AN    "DB_LIF"._x.TargIsHookunder;
      AN    "DB_LIF"._x.TargIsTop;
      AN    "DB_LIF"._x.TargIsSafety;
      A     "DB_LIF"._x.TargetSwitchPoint;
      AN    "DB_LIF"._x.TargIsLowest;
      AN    "DB_LIF"._x.TargIsIntPos;
      AN    #tmp_Targ_Man;
      O;
      AN    "DB_LIF"._x.TargIsHookover;
      AN    "DB_LIF"._x.TargIsHookunder;
      AN    "DB_LIF"._x.TargIsTop;
      AN    "DB_LIF"._x.TargIsSafety;
      AN    "DB_LIF"._x.TargetSwitchPoint;
      A     "DB_LIF"._x.TargIsLowest;
      AN    "DB_LIF"._x.TargIsIntPos;
      AN    #tmp_Targ_Man;
      O;
      AN    "DB_LIF"._x.TargIsHookover;
      AN    "DB_LIF"._x.TargIsHookunder;
      AN    "DB_LIF"._x.TargIsTop;
      AN    "DB_LIF"._x.TargIsSafety;
      AN    "DB_LIF"._x.TargetSwitchPoint;
      AN    "DB_LIF"._x.TargIsLowest;
      A     "DB_LIF"._x.TargIsIntPos;
      AN    #tmp_Targ_Man;
      O;
      AN    "DB_LIF"._x.TargIsHookover;
      AN    "DB_LIF"._x.TargIsHookunder;
      AN    "DB_LIF"._x.TargIsTop;
      AN    "DB_LIF"._x.TargIsSafety;
      AN    "DB_LIF"._x.TargetSwitchPoint;
      AN    "DB_LIF"._x.TargIsLowest;
      AN    "DB_LIF"._x.TargIsIntPos;
      A     #tmp_Targ_Man;
      );
      =     #TargetOK;
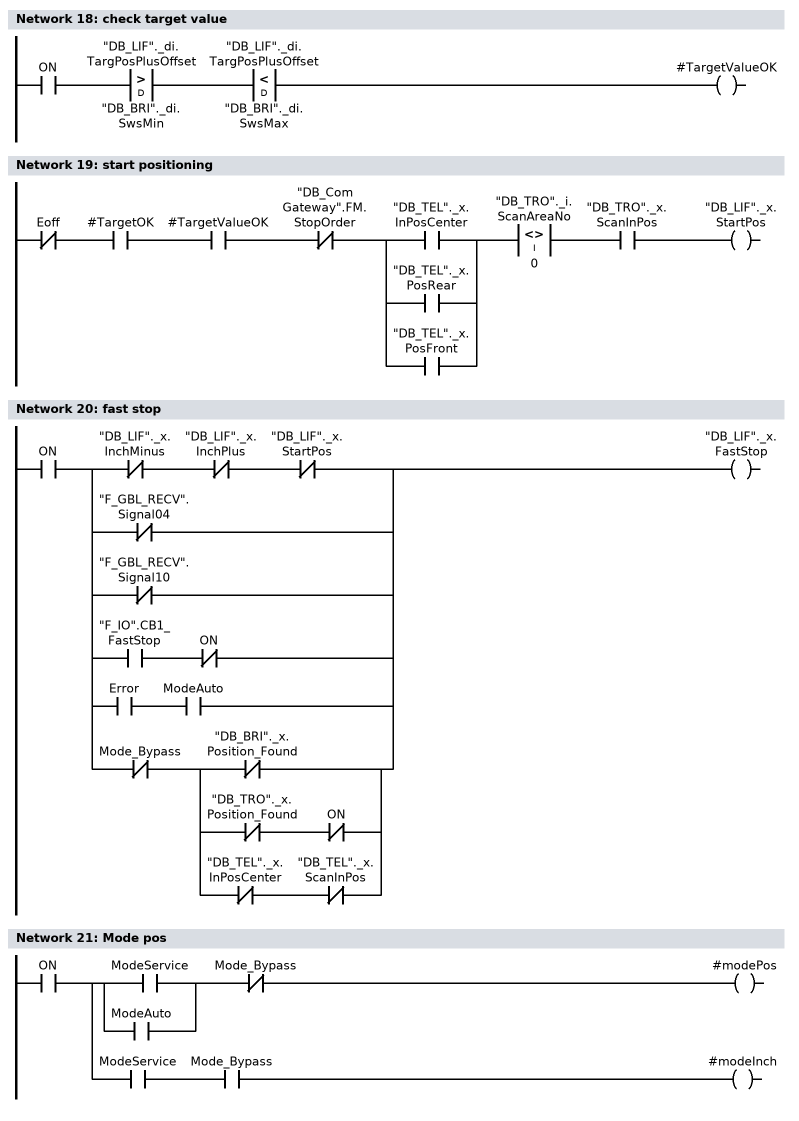
NETWORK
TITLE = check target value
      A     "ON";
      A(;
      L     "DB_LIF"._di.TargPosPlusOffset;
      L     "DB_BRI"._di.SwsMin;
      >D;
      );
      A(;
      L     "DB_LIF"._di.TargPosPlusOffset;
      L     "DB_BRI"._di.SwsMax;
      <D;
      );
      =     #TargetValueOK;
NETWORK
TITLE = start positioning
      AN    "Eoff";
      A     #TargetOK;
      A     #TargetValueOK;
      AN    "DB_ComGateway".FM.StopOrder;
      A(;
      O     "DB_TEL"._x.InPosCenter;
      O     "DB_TEL"._x.PosRear;
      O     "DB_TEL"._x.PosFront;
      );
      A(;
      L     "DB_TRO"._i.ScanAreaNo;
      L     0;
      <>I;
      );
      A     "DB_TRO"._x.ScanInPos;
      =     "DB_LIF"._x.StartPos;
NETWORK
TITLE = fast stop
      A     "ON";
      A(;
      AN    "DB_LIF"._x.InchMinus;
      AN    "DB_LIF"._x.InchPlus;
      AN    "DB_LIF"._x.StartPos;
      ON    "F_GBL_RECV".Signal04;
      ON    "F_GBL_RECV".Signal10;
      O;
      A     "F_IO".CB1_FastStop;
      AN    "ON";
      O;
      A     "Error";
      A     "ModeAuto";
      O;
      AN    "Mode_Bypass";
      A(;
      ON    "DB_BRI"._x.Position_Found;
      O;
      AN    "DB_TRO"._x.Position_Found;
      AN    "ON";
      O;
      AN    "DB_TEL"._x.InPosCenter;
      AN    "DB_TEL"._x.ScanInPos;
      );
      );
      =     "DB_LIF"._x.FastStop;
NETWORK
TITLE = Mode pos
      A     "ON";
      =     L 24.0;
      A     L 24.0;
      A(;
      O     "ModeService";
      O     "ModeAuto";
      );
      AN    "Mode_Bypass";
      =     #modePos;
      A     L 24.0;
      A     "ModeService";
      A     "Mode_Bypass";
      =     #modeInch;
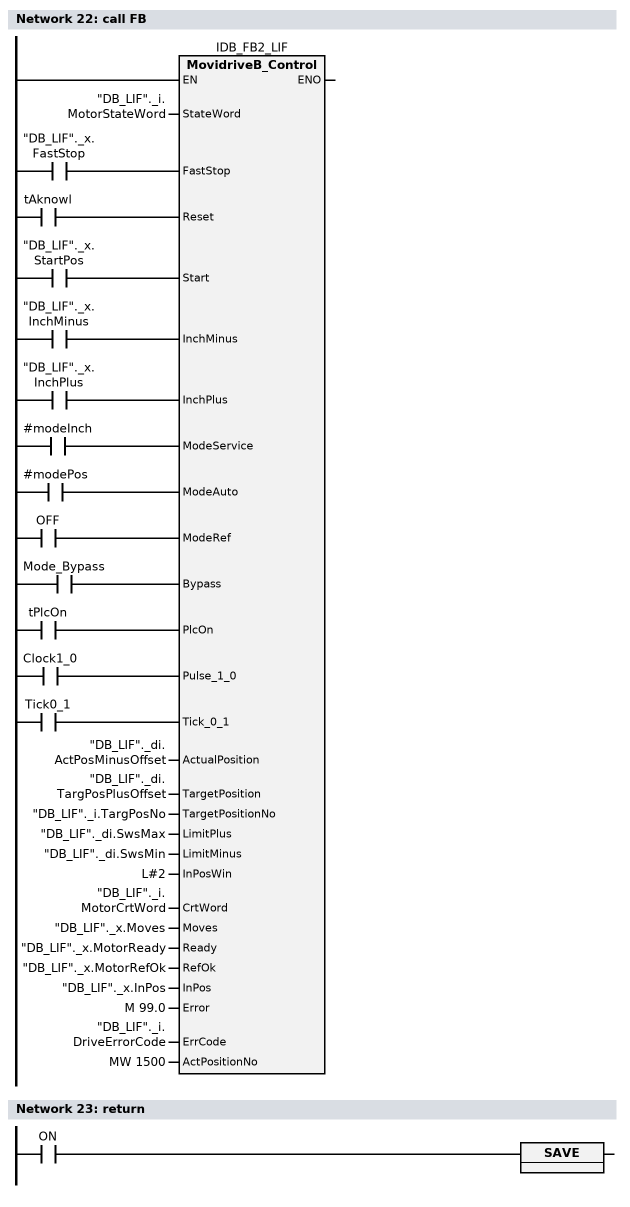
NETWORK
TITLE = call FB
      A     "DB_LIF"._x.FastStop;
      =     L 24.0;
      BLD   103;
      A     "tAknowl";
      =     L 24.1;
      BLD   103;
      A     "DB_LIF"._x.StartPos;
      =     L 24.2;
      BLD   103;
      A     "DB_LIF"._x.InchMinus;
      =     L 24.3;
      BLD   103;
      A     "DB_LIF"._x.InchPlus;
      =     L 24.4;
      BLD   103;
      A     #modeInch;
      =     L 24.5;
      BLD   103;
      A     #modePos;
      =     L 24.6;
      BLD   103;
      A     "OFF";
      =     L 24.7;
      BLD   103;
      A     "Mode_Bypass";
      =     L 25.0;
      BLD   103;
      A     "tPlcOn";
      =     L 25.1;
      BLD   103;
      A     "Clock1_0";
      =     L 25.2;
      BLD   103;
      A     "Tick0_1";
      =     L 25.3;
      BLD   103;
      CALL  "MovidriveB_Control" , "IDB_FB2_LIF" (
           StateWord                := "DB_LIF"._i.MotorStateWord,
           FastStop                 := L 24.0,
           Reset                    := L 24.1,
           Start                    := L 24.2,
           InchMinus                := L 24.3,
           InchPlus                 := L 24.4,
           ModeService              := L 24.5,
           ModeAuto                 := L 24.6,
           ModeRef                  := L 24.7,
           Bypass                   := L 25.0,
           PlcOn                    := L 25.1,
           Pulse_1_0                := L 25.2,
           Tick_0_1                 := L 25.3,
           ActualPosition           := "DB_LIF"._di.ActPosMinusOffset,
           TargetPosition           := "DB_LIF"._di.TargPosPlusOffset,
           TargetPositionNo         := "DB_LIF"._i.TargPosNo,
           LimitPlus                := "DB_LIF"._di.SwsMax,
           LimitMinus               := "DB_LIF"._di.SwsMin,
           InPosWin                 := L#2,
           CrtWord                  := "DB_LIF"._i.MotorCrtWord,
           Moves                    := "DB_LIF"._x.Moves,
           Ready                    := "DB_LIF"._x.MotorReady,
           RefOk                    := "DB_LIF"._x.MotorRefOk,
           InPos                    := "DB_LIF"._x.InPos,
           Error                    := M 99.0,
           ErrCode                  := "DB_LIF"._i.DriveErrorCode,
           ActPositionNo            := MW 1500);
      NOP   0;
NETWORK
TITLE = return
      A     "ON";
      SAVE;
END_FUNCTION

FUNCTION "Axis_LIFT_Speed" : VOID	// FC 223
TITLE = LIFT Speed
VERSION : 0.1
VAR_TEMP
  tmp_any_1 : ANY ;
  tmp_di_fs_Min : DINT ;
  tmp_di_fs_Max : DINT ;
  tmp_speed_auto : INT ;
  tmp_speed_man : INT ;
  tmp_fs2 : BOOL ;
END_VAR
BEGIN
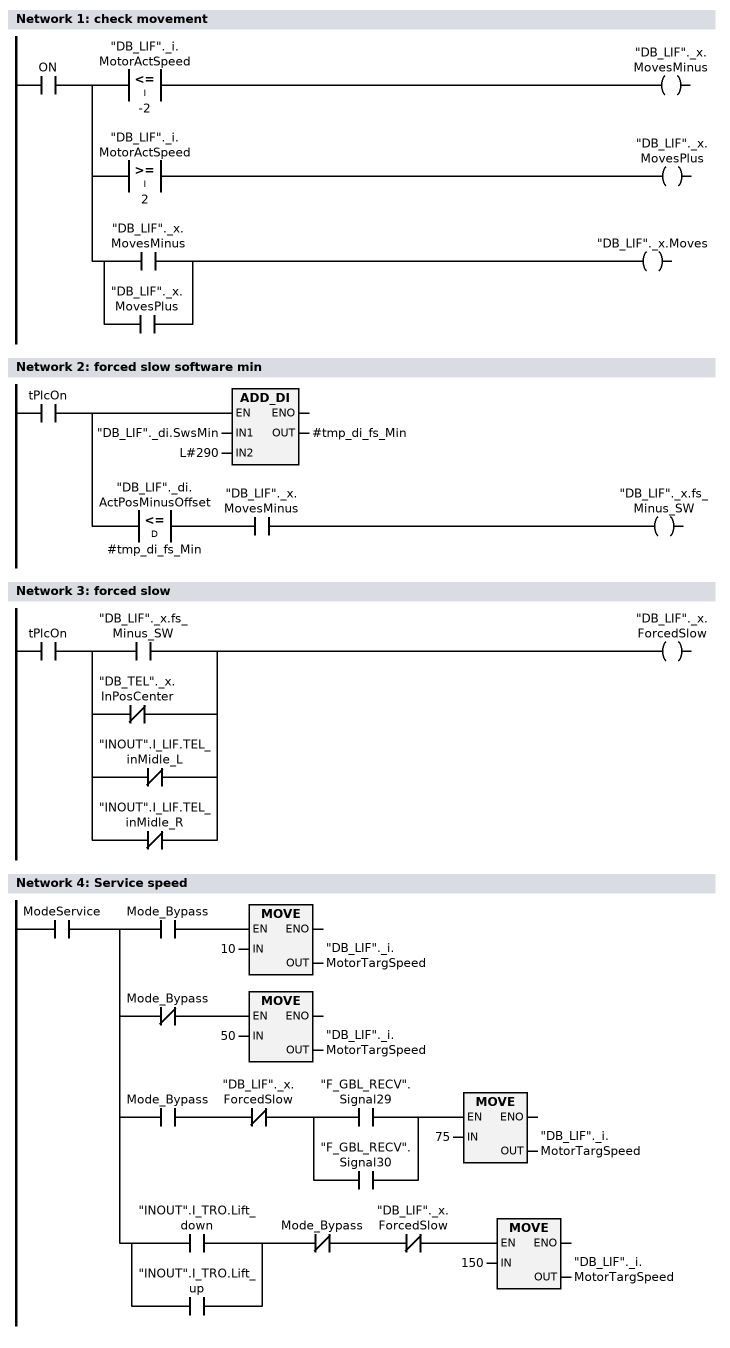
NETWORK
TITLE = check movement
      A     "ON";
      =     L 23.0;
      A     L 23.0;
      A(;
      L     "DB_LIF"._i.MotorActSpeed;
      L     -2;
      <=I;
      );
      =     "DB_LIF"._x.MovesMinus;
      A     L 23.0;
      A(;
      L     "DB_LIF"._i.MotorActSpeed;
      L     2;
      >=I;
      );
      =     "DB_LIF"._x.MovesPlus;
      A     L 23.0;
      A(;
      O     "DB_LIF"._x.MovesMinus;
      O     "DB_LIF"._x.MovesPlus;
      );
      =     "DB_LIF"._x.Moves;
NETWORK
TITLE = forced slow software min
      A     "tPlcOn";
      =     L 23.0;
      A     L 23.0;
      JNB   _001;
      L     "DB_LIF"._di.SwsMin;
      L     L#290;
      +D;
      T     #tmp_di_fs_Min;
_001: NOP   0;
      A     L 23.0;
      A(;
      L     "DB_LIF"._di.ActPosMinusOffset;
      L     #tmp_di_fs_Min;
      <=D;
      );
      A     "DB_LIF"._x.MovesMinus;
      =     "DB_LIF"._x.fs_Minus_SW;
NETWORK
TITLE = forced slow
      A     "tPlcOn";
      A(;
      O     "DB_LIF"._x.fs_Minus_SW;
      ON    "DB_TEL"._x.InPosCenter;
      ON    "INOUT".I_LIF.TEL_inMidle_L;
      ON    "INOUT".I_LIF.TEL_inMidle_R;
      );
      =     "DB_LIF"._x.ForcedSlow;
NETWORK
TITLE = Service speed
//fast speed only if telescope in middle pos 75
      A     "ModeService";
      =     L 23.0;
      A     L 23.0;
      A     "Mode_Bypass";
      JNB   _002;
      L     10;
      T     "DB_LIF"._i.MotorTargSpeed;
_002: NOP   0;
      A     L 23.0;
      AN    "Mode_Bypass";
      JNB   _003;
      L     50;
      T     "DB_LIF"._i.MotorTargSpeed;
_003: NOP   0;
      A     L 23.0;
      A     "Mode_Bypass";
      AN    "DB_LIF"._x.ForcedSlow;
      A(;
      O     "F_GBL_RECV".Signal29;
      O     "F_GBL_RECV".Signal30;
      );
      JNB   _004;
      L     75;
      T     "DB_LIF"._i.MotorTargSpeed;
_004: NOP   0;
      A     L 23.0;
      A(;
      O     "INOUT".I_TRO.Lift_down;
      O     "INOUT".I_TRO.Lift_up;
      );
      AN    "Mode_Bypass";
      AN    "DB_LIF"._x.ForcedSlow;
      JNB   _005;
      L     150;
      T     "DB_LIF"._i.MotorTargSpeed;
_005: NOP   0;
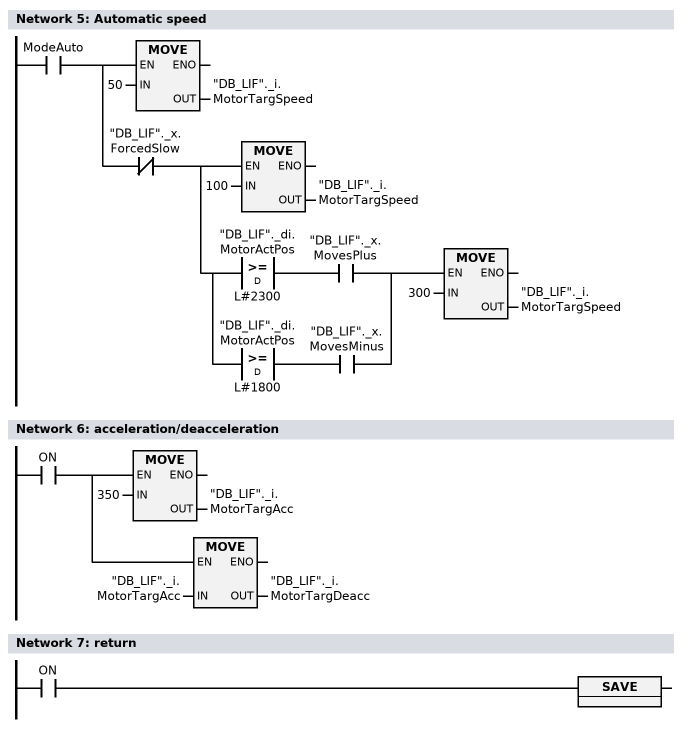
NETWORK
TITLE = Automatic speed
//fast speed only if telescope in middle pos
//Slower speed in transition from RBG to rack 450
      A     "ModeAuto";
      =     L 23.0;
      A     L 23.0;
      JNB   _006;
      L     50;
      T     "DB_LIF"._i.MotorTargSpeed;
_006: NOP   0;
      A     L 23.0;
      AN    "DB_LIF"._x.ForcedSlow;
      =     L 23.1;
      A     L 23.1;
      JNB   _007;
      L     100;
      T     "DB_LIF"._i.MotorTargSpeed;
_007: NOP   0;
      A     L 23.1;
      A(;
      A(;
      L     "DB_LIF"._di.MotorActPos;
      L     L#2300;
      >=D;
      );
      A     "DB_LIF"._x.MovesPlus;
      O;
      A(;
      L     "DB_LIF"._di.MotorActPos;
      L     L#1800;
      >=D;
      );
      A     "DB_LIF"._x.MovesMinus;
      );
      JNB   _008;
      L     300;
      T     "DB_LIF"._i.MotorTargSpeed;
_008: NOP   0;
NETWORK
TITLE = acceleration/deacceleration
      A     "ON";
      =     L 23.0;
      A     L 23.0;
      JNB   _009;
      L     350;
      T     "DB_LIF"._i.MotorTargAcc;
_009: NOP   0;
      A     L 23.0;
      JNB   _00a;
      L     "DB_LIF"._i.MotorTargAcc;
      T     "DB_LIF"._i.MotorTargDeacc;
_00a: NOP   0;
NETWORK
TITLE = return
      A     "ON";
      SAVE;
END_FUNCTION

FUNCTION "Axis_LIFT_Scan" : VOID	// FC 224
TITLE = LIFT scan positions
VERSION : 0.1
VAR_TEMP
  tmpHookDataSet : UDT 102;
  tmp_di_posValHO : DINT ;
  tmp_di_posValHU : DINT ;
  tmp_di_1 : DINT ;
  winDiff : DINT ;
  tmp_di_StpWin : DINT ;
  tmp_di_PosWin : DINT ;
  RetVal : INT ;
  winOK : BOOL ;
  tmp_inPosTopChk : BOOL ;
  tmp_inPosTopStp : BOOL ;
  tmp_inPos : BOOL ;
  tmp_auto_target_right : BOOL ;
  tmp_direction_right : BOOL ;
  top_set : BOOL ;
  top_rset : BOOL ;
  tmp_offset : INT ;
  tmp_DIR : BOOL ;
END_VAR
BEGIN
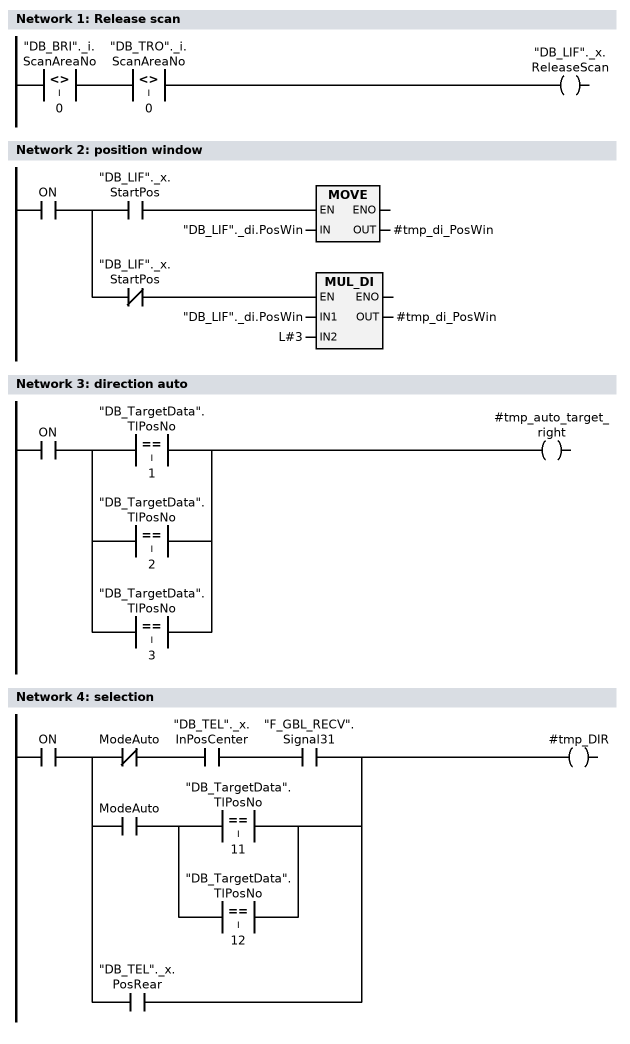
NETWORK
TITLE = Release scan
//scan always if a area is avaiable
      A(;
      L     "DB_BRI"._i.ScanAreaNo;
      L     0;
      <>I;
      );
      A(;
      L     "DB_TRO"._i.ScanAreaNo;
      L     0;
      <>I;
      );
      =     "DB_LIF"._x.ReleaseScan;
NETWORK
TITLE = position window
      A     "ON";
      =     L 87.0;
      A     L 87.0;
      A     "DB_LIF"._x.StartPos;
      JNB   _001;
      L     "DB_LIF"._di.PosWin;
      T     #tmp_di_PosWin;
_001: NOP   0;
      A     L 87.0;
      AN    "DB_LIF"._x.StartPos;
      JNB   _002;
      L     "DB_LIF"._di.PosWin;
      L     L#3;
      *D;
      T     #tmp_di_PosWin;
_002: NOP   0;
NETWORK
TITLE = direction auto
      A     "ON";
      A(;
      O(;
      L     "DB_TargetData".TlPosNo;
      L     1;
      ==I;
      );
      O(;
      L     "DB_TargetData".TlPosNo;
      L     2;
      ==I;
      );
      O(;
      L     "DB_TargetData".TlPosNo;
      L     3;
      ==I;
      );
      );
      =     #tmp_auto_target_right;
NETWORK
TITLE = selection
      A     "ON";
      A(;
      AN    "ModeAuto";
      A     "DB_TEL"._x.InPosCenter;
      A     "F_GBL_RECV".Signal31;
      O;
      A     "ModeAuto";
      A(;
      O(;
      L     "DB_TargetData".TlPosNo;
      L     11;
      ==I;
      );
      O(;
      L     "DB_TargetData".TlPosNo;
      L     12;
      ==I;
      );
      );
      O     "DB_TEL"._x.PosRear;
      );
      =     #tmp_DIR;
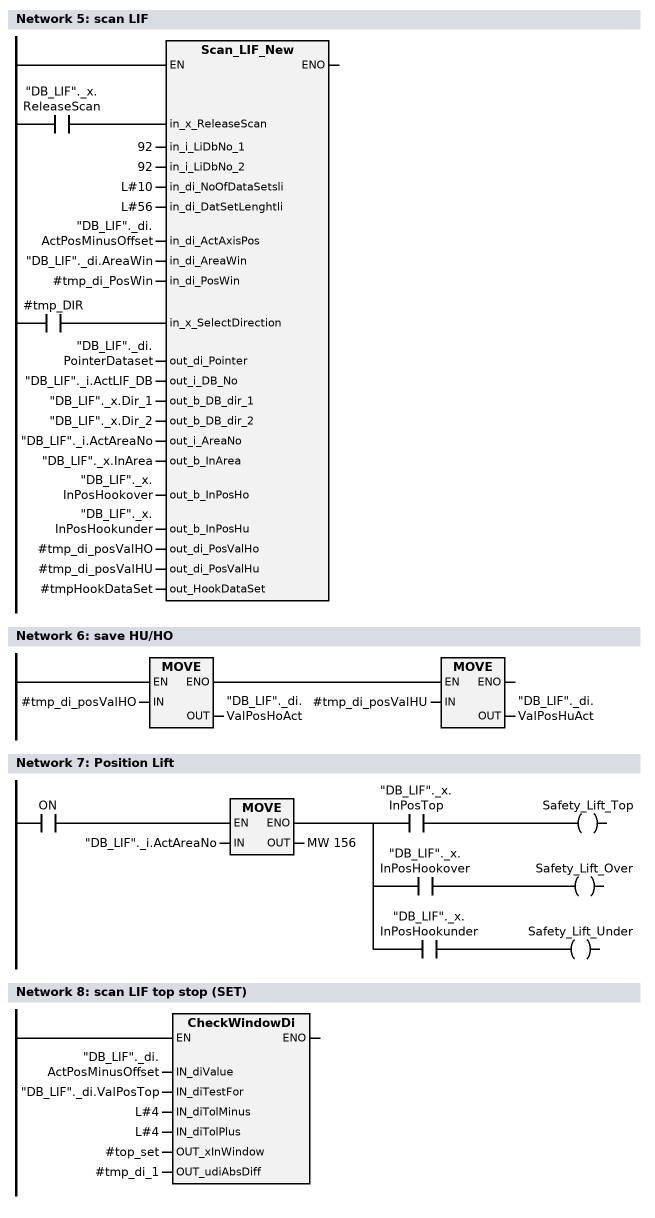
NETWORK
TITLE = scan LIF
//"DB_LIF"._i.ActLiDbNo_1 an 92
//"DB_LIF"._i.ActLiDbNo_2 an 93
      A     "DB_LIF"._x.ReleaseScan;
      =     L 87.0;
      BLD   103;
      A     #tmp_DIR;
      =     L 87.1;
      BLD   103;
      CALL  "Scan_LIF_New" (
           in_x_ReleaseScan         := L 87.0,
           in_i_LiDbNo_1            := 92,
           in_i_LiDbNo_2            := 92,
           in_di_NoOfDataSetsli     := L#10,
           in_di_DatSetLenghtli     := L#56,
           in_di_ActAxisPos         := "DB_LIF"._di.ActPosMinusOffset,
           in_di_AreaWin            := "DB_LIF"._di.AreaWin,
           in_di_PosWin             := #tmp_di_PosWin,
           in_x_SelectDirection     := L 87.1,
           out_di_Pointer           := "DB_LIF"._di.PointerDataset,
           out_i_DB_No              := "DB_LIF"._i.ActLIF_DB,
           out_b_DB_dir_1           := "DB_LIF"._x.Dir_1,
           out_b_DB_dir_2           := "DB_LIF"._x.Dir_2,
           out_i_AreaNo             := "DB_LIF"._i.ActAreaNo,
           out_b_InArea             := "DB_LIF"._x.InArea,
           out_b_InPosHo            := "DB_LIF"._x.InPosHookover,
           out_b_InPosHu            := "DB_LIF"._x.InPosHookunder,
           out_di_PosValHo          := #tmp_di_posValHO,
           out_di_PosValHu          := #tmp_di_posValHU,
           out_HookDataSet          := #tmpHookDataSet);
      NOP   0;
NETWORK
TITLE = save HU/HO
      A(;
      L     #tmp_di_posValHO;
      T     "DB_LIF"._di.ValPosHoAct;
      SET;
      SAVE;
      CLR;
      A     BR;
      );
      JNB   _003;
      L     #tmp_di_posValHU;
      T     "DB_LIF"._di.ValPosHuAct;
_003: NOP   0;
NETWORK
TITLE = Position Lift
      A     "ON";
      JNB   _004;
      L     "DB_LIF"._i.ActAreaNo;
      T     MW 156;
      SET;
      SAVE;
      CLR;
_004: A     BR;
      =     L 87.0;
      A     L 87.0;
      A     "DB_LIF"._x.InPosTop;
      =     "Safety_Lift_Top";
      A     L 87.0;
      A     "DB_LIF"._x.InPosHookover;
      =     "Safety_Lift_Over";
      A     L 87.0;
      A     "DB_LIF"._x.InPosHookunder;
      =     "Safety_Lift_Under";
NETWORK
TITLE = scan LIF top stop (SET)
//The position is on the laser 278, but in the software 342. SEW scaling is 
//incorrect 
      CALL  "CheckWindowDi" (
           IN_diValue               := "DB_LIF"._di.ActPosMinusOffset,
           IN_diTestFor             := "DB_LIF"._di.ValPosTop,
           IN_diTolMinus            := L#4,
           IN_diTolPlus             := L#4,
           OUT_xInWindow            := #top_set,
           OUT_udiAbsDiff           := #tmp_di_1);
      NOP   0;
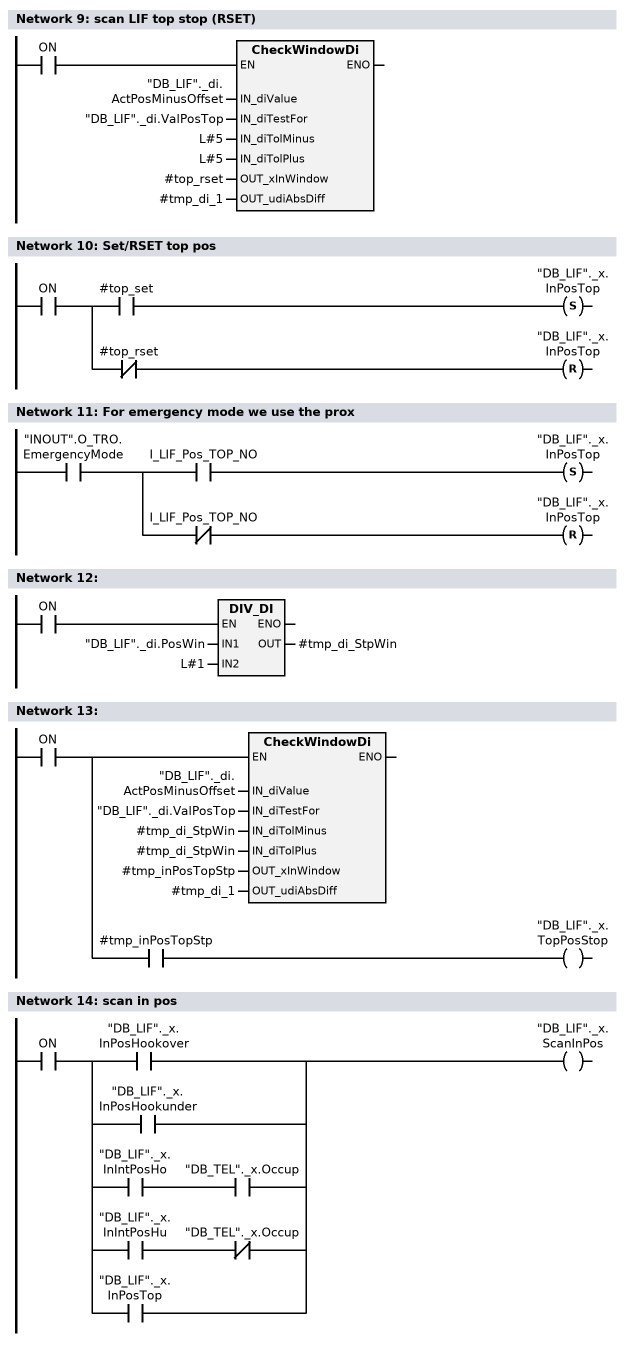
NETWORK
TITLE = scan LIF top stop (RSET)
      A     "ON";
      JNB   _005;
      CALL  "CheckWindowDi" (
           IN_diValue               := "DB_LIF"._di.ActPosMinusOffset,
           IN_diTestFor             := "DB_LIF"._di.ValPosTop,
           IN_diTolMinus            := L#5,
           IN_diTolPlus             := L#5,
           OUT_xInWindow            := #top_rset,
           OUT_udiAbsDiff           := #tmp_di_1);
_005: NOP   0;
NETWORK
TITLE = Set/RSET top pos
      A     "ON";
      =     L 87.0;
      A     L 87.0;
      A     #top_set;
      S     "DB_LIF"._x.InPosTop;
      A     L 87.0;
      AN    #top_rset;
      R     "DB_LIF"._x.InPosTop;
NETWORK
TITLE = For emergency mode we use the prox
      A     "INOUT".O_TRO.EmergencyMode;
      =     L 87.0;
      A     L 87.0;
      A     "I_LIF_Pos_TOP_NO";
      S     "DB_LIF"._x.InPosTop;
      A     L 87.0;
      AN    "I_LIF_Pos_TOP_NO";
      R     "DB_LIF"._x.InPosTop;
NETWORK
TITLE =
      A     "ON";
      JNB   _006;
      L     "DB_LIF"._di.PosWin;
      L     L#1;
      /D;
      T     #tmp_di_StpWin;
_006: NOP   0;
NETWORK
TITLE =
      A     "ON";
      =     L 87.0;
      A     L 87.0;
      JNB   _007;
      CALL  "CheckWindowDi" (
           IN_diValue               := "DB_LIF"._di.ActPosMinusOffset,
           IN_diTestFor             := "DB_LIF"._di.ValPosTop,
           IN_diTolMinus            := #tmp_di_StpWin,
           IN_diTolPlus             := #tmp_di_StpWin,
           OUT_xInWindow            := #tmp_inPosTopStp,
           OUT_udiAbsDiff           := #tmp_di_1);
_007: NOP   0;
      A     L 87.0;
      A     #tmp_inPosTopStp;
      =     "DB_LIF"._x.TopPosStop;
NETWORK
TITLE = scan in pos
      A     "ON";
      A(;
      O     "DB_LIF"._x.InPosHookover;
      O     "DB_LIF"._x.InPosHookunder;
      O;
      A     "DB_LIF"._x.InIntPosHo;
      A     "DB_TEL"._x.Occup;
      O;
      A     "DB_LIF"._x.InIntPosHu;
      AN    "DB_TEL"._x.Occup;
      O     "DB_LIF"._x.InPosTop;
      );
      =     "DB_LIF"._x.ScanInPos;
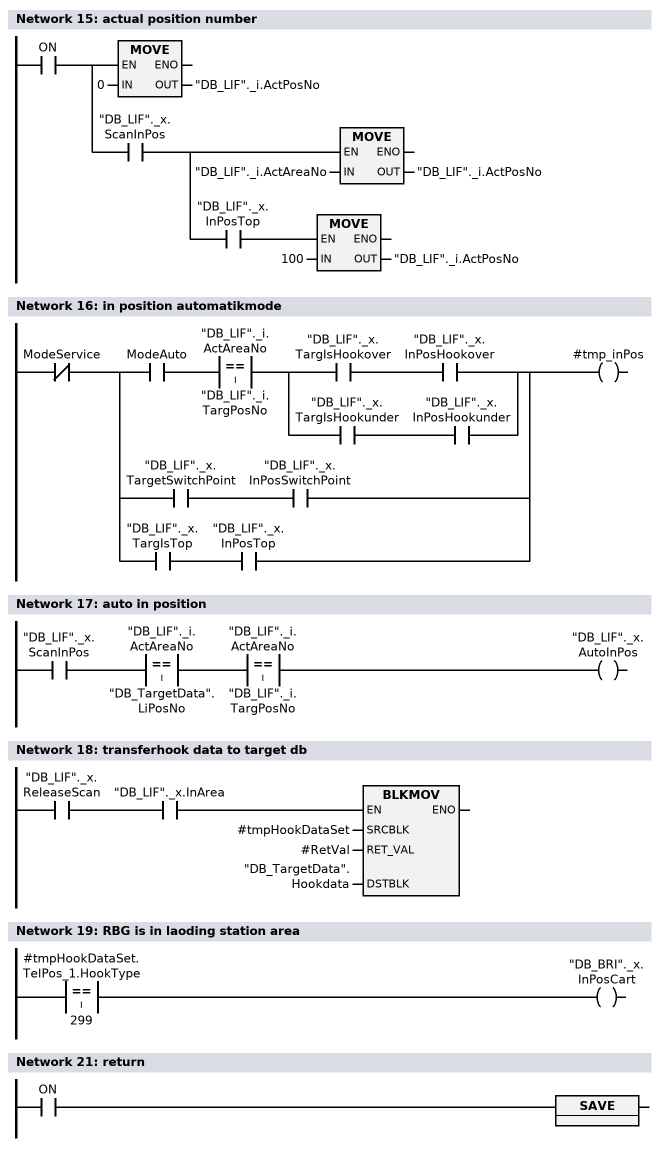
NETWORK
TITLE = actual position number
      A     "ON";
      =     L 87.0;
      A     L 87.0;
      JNB   _008;
      L     0;
      T     "DB_LIF"._i.ActPosNo;
_008: NOP   0;
      A     L 87.0;
      A     "DB_LIF"._x.ScanInPos;
      =     L 87.1;
      A     L 87.1;
      JNB   _009;
      L     "DB_LIF"._i.ActAreaNo;
      T     "DB_LIF"._i.ActPosNo;
_009: NOP   0;
      A     L 87.1;
      A     "DB_LIF"._x.InPosTop;
      JNB   _00a;
      L     100;
      T     "DB_LIF"._i.ActPosNo;
_00a: NOP   0;
NETWORK
TITLE = in position automatikmode 
      AN    "ModeService";
      A(;
      A     "ModeAuto";
      A(;
      L     "DB_LIF"._i.ActAreaNo;
      L     "DB_LIF"._i.TargPosNo;
      ==I;
      );
      A(;
      A     "DB_LIF"._x.TargIsHookover;
      A     "DB_LIF"._x.InPosHookover;
      O;
      A     "DB_LIF"._x.TargIsHookunder;
      A     "DB_LIF"._x.InPosHookunder;
      );
      O;
      A     "DB_LIF"._x.TargetSwitchPoint;
      A     "DB_LIF"._x.InPosSwitchPoint;
      O;
      A     "DB_LIF"._x.TargIsTop;
      A     "DB_LIF"._x.InPosTop;
      );
      =     #tmp_inPos;
NETWORK
TITLE = auto in position
      A     "DB_LIF"._x.ScanInPos;
      A(;
      L     "DB_LIF"._i.ActAreaNo;
      L     "DB_TargetData".LiPosNo;
      ==I;
      );
      A(;
      L     "DB_LIF"._i.ActAreaNo;
      L     "DB_LIF"._i.TargPosNo;
      ==I;
      );
      =     "DB_LIF"._x.AutoInPos;
NETWORK
TITLE = transferhook data to target db
      A     "DB_LIF"._x.ReleaseScan;
      A     "DB_LIF"._x.InArea;
      JNB   _00b;
      CALL  "BLKMOV" (
           SRCBLK                   := #tmpHookDataSet,
           RET_VAL                  := #RetVal,
           DSTBLK                   := "DB_TargetData".Hookdata);
_00b: NOP   0;
NETWORK
TITLE = RBG is in laoding station area
      L     #tmpHookDataSet.TelPos_1.HookType;
      L     299;
      ==I;
      =     "DB_BRI"._x.InPosCart;
NETWORK
TITLE = power control measure diameter
NETWORK
TITLE = return
      A     "ON";
      SAVE;
END_FUNCTION

FUNCTION "Axis_LIFT_Flt_081-096" : VOID	// FC 229
TITLE = Error Lift 81-96
VERSION : 0.1
BEGIN
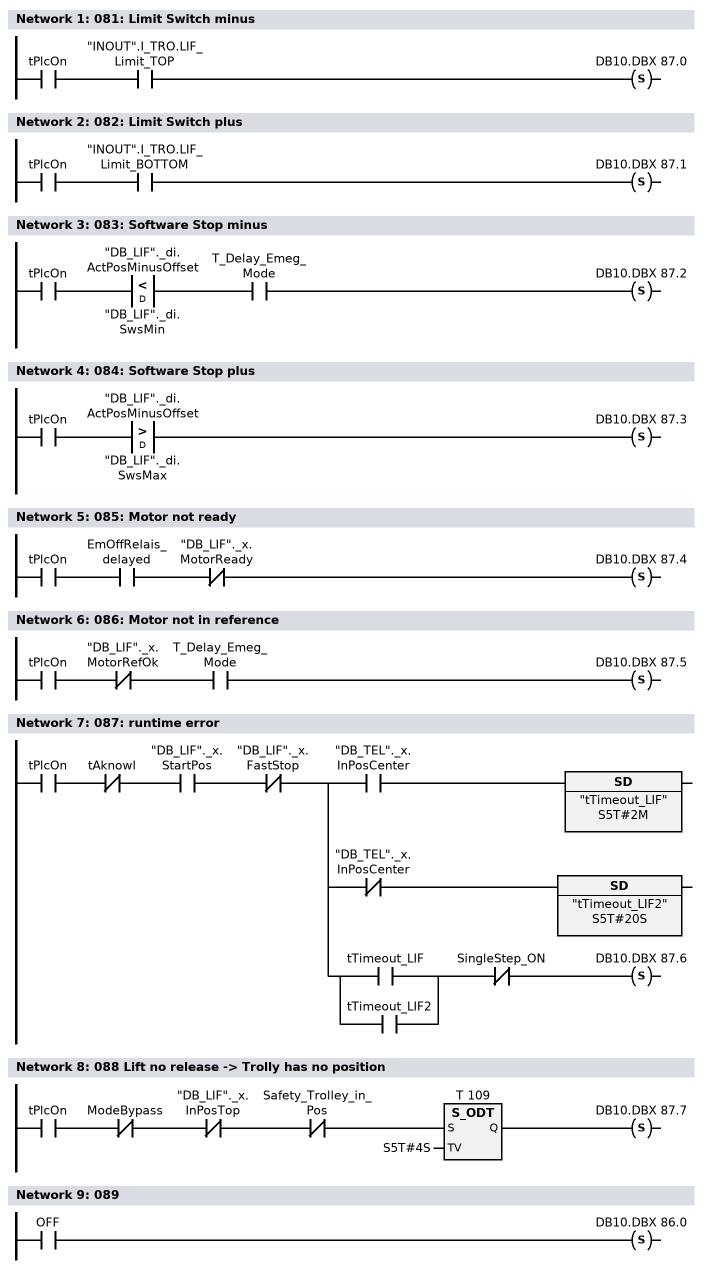
NETWORK
TITLE = 081: Limit Switch minus
      A     "tPlcOn";
      A     "INOUT".I_TRO.LIF_Limit_TOP;
      S     DB10.DBX 87.0;
NETWORK
TITLE = 082: Limit Switch plus
      A     "tPlcOn";
      A     "INOUT".I_TRO.LIF_Limit_BOTTOM;
      S     DB10.DBX 87.1;
NETWORK
TITLE = 083: Software Stop minus
      A     "tPlcOn";
      A(;
      L     "DB_LIF"._di.ActPosMinusOffset;
      L     "DB_LIF"._di.SwsMin;
      <D;
      );
      A     "T_Delay_Emeg_Mode";
      S     DB10.DBX 87.2;
NETWORK
TITLE = 084: Software Stop plus
      A     "tPlcOn";
      A(;
      L     "DB_LIF"._di.ActPosMinusOffset;
      L     "DB_LIF"._di.SwsMax;
      >D;
      );
      S     DB10.DBX 87.3;
NETWORK
TITLE = 085: Motor not ready
      A     "tPlcOn";
      A     "EmOffRelais_delayed";
      AN    "DB_LIF"._x.MotorReady;
      S     DB10.DBX 87.4;
NETWORK
TITLE = 086: Motor not in reference
      A     "tPlcOn";
      AN    "DB_LIF"._x.MotorRefOk;
      A     "T_Delay_Emeg_Mode";
      S     DB10.DBX 87.5;
NETWORK
TITLE = 087: runtime error
      A     "tPlcOn";
      AN    "tAknowl";
      A     "DB_LIF"._x.StartPos;
      AN    "DB_LIF"._x.FastStop;
      =     L 0.0;
      A     L 0.0;
      A     "DB_TEL"._x.InPosCenter;
      L     S5T#2M;
      SD    "tTimeout_LIF";
      A     L 0.0;
      AN    "DB_TEL"._x.InPosCenter;
      L     S5T#20S;
      SD    "tTimeout_LIF2";
      A     L 0.0;
      A(;
      O     "tTimeout_LIF";
      O     "tTimeout_LIF2";
      );
      AN    "SingleStep_ON";
      S     DB10.DBX 87.6;
NETWORK
TITLE = 088 Lift no release -> Trolly has no position
//07 Sensor forced slow minus
      A     "tPlcOn";
      AN    "ModeBypass";
      AN    "DB_LIF"._x.InPosTop;
      AN    "Safety_Trolley_in_Pos";
      L     S5T#4S;
      SD    T 109;
      NOP   0;
      NOP   0;
      NOP   0;
      A     T 109;
      S     DB10.DBX 87.7;
NETWORK
TITLE = 089
//08 Sensor forced slow plus
      A     "OFF";
      S     DB10.DBX 86.0;
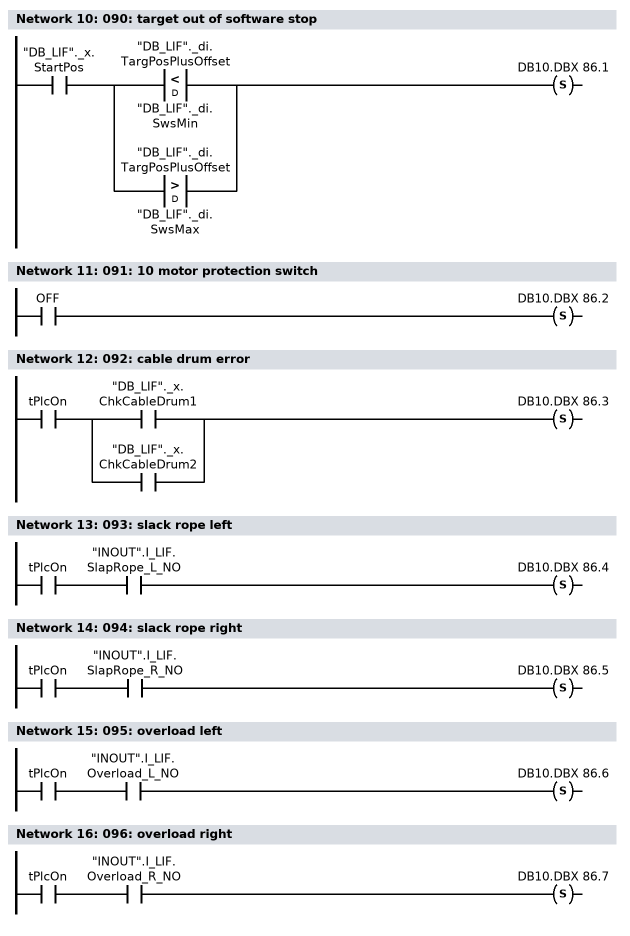
NETWORK
TITLE = 090: target out of software stop
      A     "DB_LIF"._x.StartPos;
      A(;
      O(;
      L     "DB_LIF"._di.TargPosPlusOffset;
      L     "DB_LIF"._di.SwsMin;
      <D;
      );
      O(;
      L     "DB_LIF"._di.TargPosPlusOffset;
      L     "DB_LIF"._di.SwsMax;
      >D;
      );
      );
      S     DB10.DBX 86.1;
NETWORK
TITLE = 091: 10 motor protection switch
      A     "OFF";
      S     DB10.DBX 86.2;
NETWORK
TITLE = 092: cable drum error
      A     "tPlcOn";
      A(;
      O     "DB_LIF"._x.ChkCableDrum1;
      O     "DB_LIF"._x.ChkCableDrum2;
      );
      S     DB10.DBX 86.3;
NETWORK
TITLE = 093: slack rope left
      A     "tPlcOn";
      A     "INOUT".I_LIF.SlapRope_L_NO;
      S     DB10.DBX 86.4;
NETWORK
TITLE = 094: slack rope right
      A     "tPlcOn";
      A     "INOUT".I_LIF.SlapRope_R_NO;
      S     DB10.DBX 86.5;
NETWORK
TITLE = 095: overload left
      A     "tPlcOn";
      A     "INOUT".I_LIF.Overload_L_NO;
      S     DB10.DBX 86.6;
NETWORK
TITLE = 096: overload right
      A     "tPlcOn";
      A     "INOUT".I_LIF.Overload_R_NO;
      S     DB10.DBX 86.7;
END_FUNCTION

FUNCTION "Axis_TELESCOPES" : VOID	// FC 230
TITLE = Axis TELESCOPES
VERSION : 0.1
BEGIN
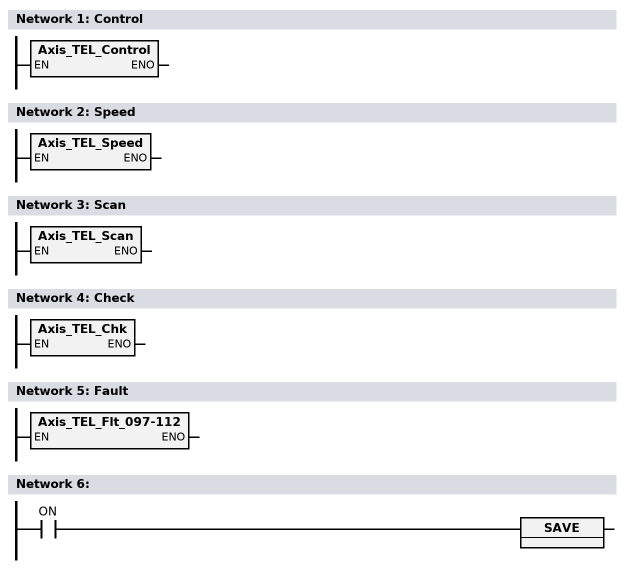
NETWORK
TITLE = Control
      CALL  "Axis_TEL_Control";
      NOP   0;
NETWORK
TITLE = Speed
      CALL  "Axis_TEL_Speed";
      NOP   0;
NETWORK
TITLE = Scan
      CALL  "Axis_TEL_Scan";
      NOP   0;
NETWORK
TITLE = Check
      CALL  "Axis_TEL_Chk";
      NOP   0;
NETWORK
TITLE = Fault
      CALL  "Axis_TEL_Flt_097-112";
      NOP   0;
NETWORK
TITLE =
      A     "ON";
      SAVE;
END_FUNCTION

FUNCTION "Axis_TEL_Control" : VOID	// FC 232
TITLE = Axis TELESCOPES Control
VERSION : 0.1
VAR_TEMP
  tmp_di_PosWindow : DINT ;
  tmp_di_StopWindow : DINT ;
  tmpAutoCenter : BOOL ;
  tmpManCenterMinus : BOOL ;
  tmpManCenterPlus : BOOL ;
  tmp_fastspeed : BOOL ;
  tmp_TargetHook_Auto : BOOL ;
  tmp_TargetHook_Manual : BOOL ;
  tmp_TargetValueOK : BOOL ;
  tmp_release : BOOL ;
  tmp_ValPosMin : DINT ;
  tmp_ValPosMax : DINT ;
  mode_ref : BOOL ;
  InPos : BOOL ;
  Target_Ok : BOOL ;
  tmpInAreaLS1 : BOOL ;
  tmpInAreaLS2 : BOOL ;
  tmpInAreaLS3 : BOOL ;
  tmpInAreaRack : BOOL ;
  relSize : BOOL ;
  target_lomg_1 : BOOL ;
  target_short_1 : BOOL ;
  target_short_2 : BOOL ;
  target_long_11 : BOOL ;
  target_short_11 : BOOL ;
  target_short_12 : BOOL ;
END_VAR
BEGIN
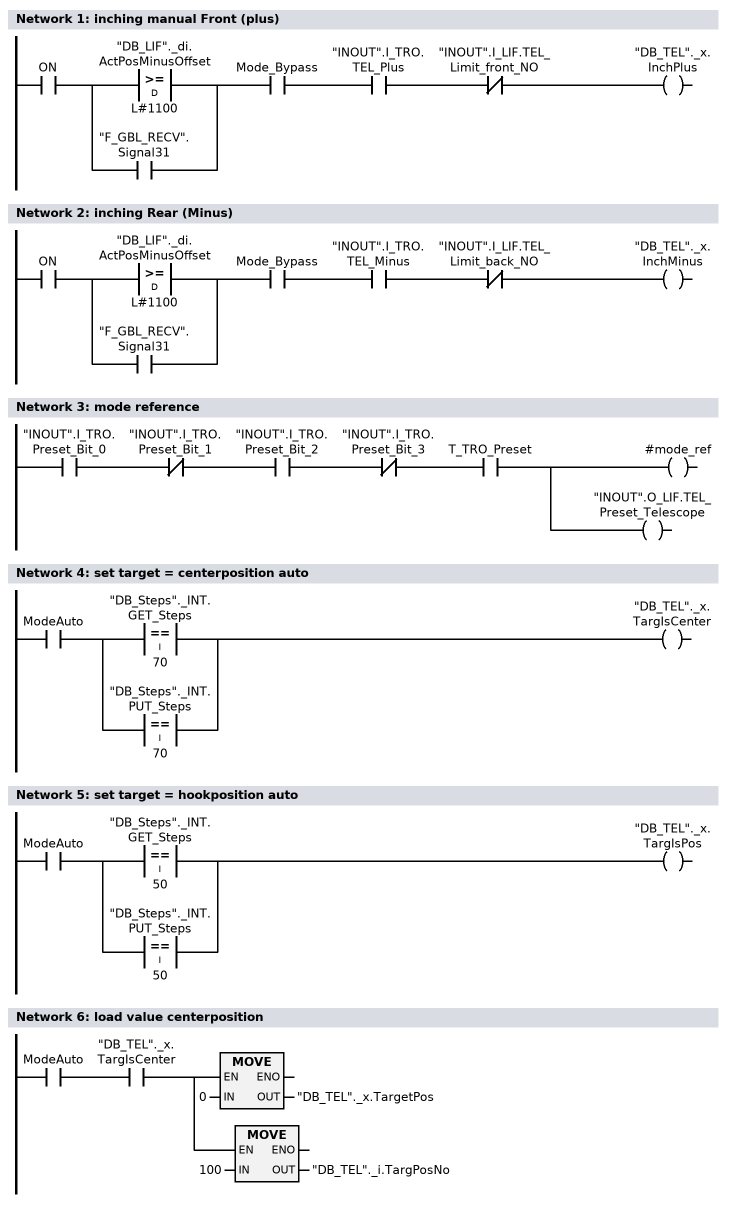
NETWORK
TITLE = inching manual Front (plus)
      A     "ON";
      A(;
      O(;
      L     "DB_LIF"._di.ActPosMinusOffset;
      L     L#1100;
      >=D;
      );
      O     "F_GBL_RECV".Signal31;
      );
      A     "Mode_Bypass";
      A     "INOUT".I_TRO.TEL_Plus;
      AN    "INOUT".I_LIF.TEL_Limit_front_NO;
      =     "DB_TEL"._x.InchPlus;
NETWORK
TITLE = inching Rear (Minus)
      A     "ON";
      A(;
      O(;
      L     "DB_LIF"._di.ActPosMinusOffset;
      L     L#1100;
      >=D;
      );
      O     "F_GBL_RECV".Signal31;
      );
      A     "Mode_Bypass";
      A     "INOUT".I_TRO.TEL_Minus;
      AN    "INOUT".I_LIF.TEL_Limit_back_NO;
      =     "DB_TEL"._x.InchMinus;
NETWORK
TITLE = mode reference
      A     "INOUT".I_TRO.Preset_Bit_0;
      AN    "INOUT".I_TRO.Preset_Bit_1;
      A     "INOUT".I_TRO.Preset_Bit_2;
      AN    "INOUT".I_TRO.Preset_Bit_3;
      A     "T_TRO_Preset";
      =     #mode_ref;
      =     "INOUT".O_LIF.TEL_Preset_Telescope;
NETWORK
TITLE = set target = centerposition auto
      A     "ModeAuto";
      A(;
      O(;
      L     "DB_Steps"._INT.GET_Steps;
      L     70;
      ==I;
      );
      O(;
      L     "DB_Steps"._INT.PUT_Steps;
      L     70;
      ==I;
      );
      );
      =     "DB_TEL"._x.TargIsCenter;
NETWORK
TITLE = set target = hookposition auto
      A     "ModeAuto";
      A(;
      O(;
      L     "DB_Steps"._INT.GET_Steps;
      L     50;
      ==I;
      );
      O(;
      L     "DB_Steps"._INT.PUT_Steps;
      L     50;
      ==I;
      );
      );
      =     "DB_TEL"._x.TargIsPos;
NETWORK
TITLE = load value centerposition
      A     "ModeAuto";
      A     "DB_TEL"._x.TargIsCenter;
      =     L 20.0;
      A     L 20.0;
      JNB   _001;
      L     0;
      T     "DB_TEL"._x.TargetPos;
_001: NOP   0;
      A     L 20.0;
      JNB   _002;
      L     100;
      T     "DB_TEL"._i.TargPosNo;
_002: NOP   0;
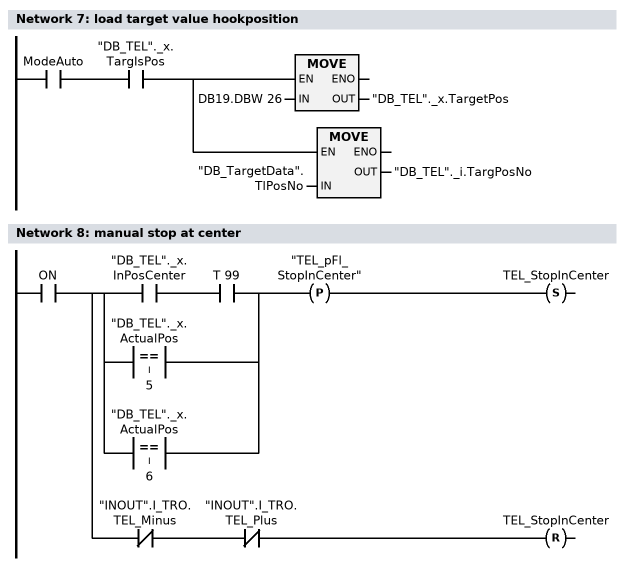
NETWORK
TITLE = load target value hookposition 
      A     "ModeAuto";
      A     "DB_TEL"._x.TargIsPos;
      =     L 20.0;
      A     L 20.0;
      JNB   _003;
      L     DB19.DBW 26;
      T     "DB_TEL"._x.TargetPos;
_003: NOP   0;
      A     L 20.0;
      JNB   _004;
      L     "DB_TargetData".TlPosNo;
      T     "DB_TEL"._i.TargPosNo;
_004: NOP   0;
NETWORK
TITLE = manual stop at center
      A     "ON";
      =     L 20.0;
      A     L 20.0;
      A(;
      A     "DB_TEL"._x.InPosCenter;
      A     T 99;
      O(;
      L     "DB_TEL"._x.ActualPos;
      L     5;
      ==I;
      );
      O(;
      L     "DB_TEL"._x.ActualPos;
      L     6;
      ==I;
      );
      );
      FP    "TEL_pFl_StopInCenter";
      S     "TEL_StopInCenter";
      A     L 20.0;
      AN    "INOUT".I_TRO.TEL_Minus;
      AN    "INOUT".I_TRO.TEL_Plus;
      R     "TEL_StopInCenter";
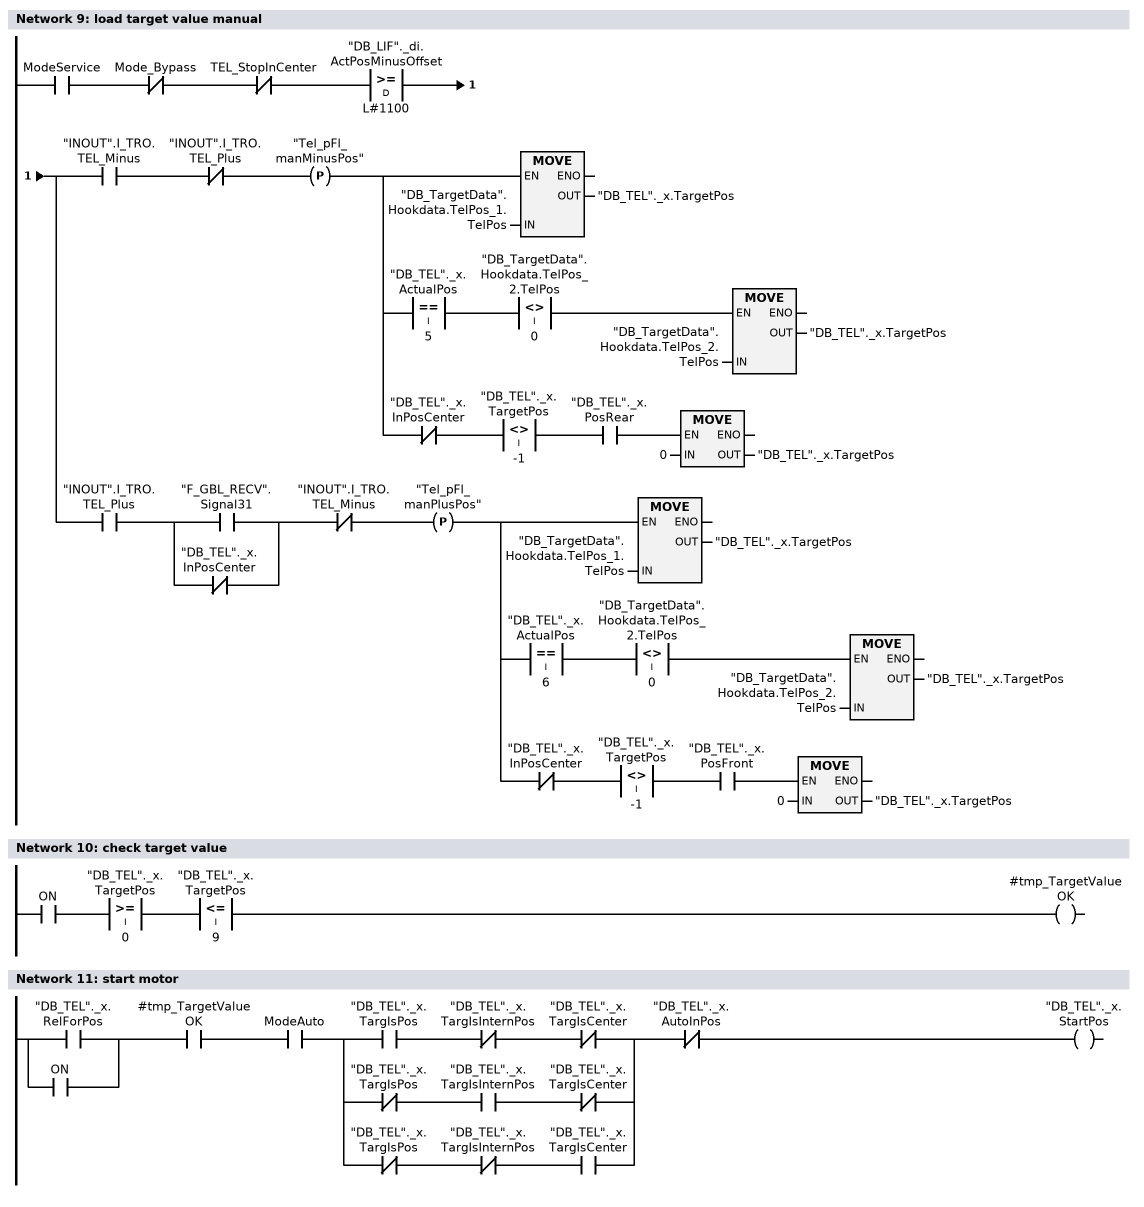
NETWORK
TITLE = load target value manual
      A     "ModeService";
      AN    "Mode_Bypass";
      AN    "TEL_StopInCenter";
      A(;
      L     "DB_LIF"._di.ActPosMinusOffset;
      L     L#1100;
      >=D;
      );
      =     L 20.0;
      A     L 20.0;
      A     "INOUT".I_TRO.TEL_Minus;
      AN    "INOUT".I_TRO.TEL_Plus;
      FP    "Tel_pFl_manMinusPos";
      =     L 20.1;
      A     L 20.1;
      JNB   _005;
      L     "DB_TargetData".Hookdata.TelPos_1.TelPos;
      T     "DB_TEL"._x.TargetPos;
_005: NOP   0;
      A     L 20.1;
      A(;
      L     "DB_TEL"._x.ActualPos;
      L     5;
      ==I;
      );
      A(;
      L     "DB_TargetData".Hookdata.TelPos_2.TelPos;
      L     0;
      <>I;
      );
      JNB   _006;
      L     "DB_TargetData".Hookdata.TelPos_2.TelPos;
      T     "DB_TEL"._x.TargetPos;
_006: NOP   0;
      A     L 20.1;
      AN    "DB_TEL"._x.InPosCenter;
      A(;
      L     "DB_TEL"._x.TargetPos;
      L     -1;
      <>I;
      );
      A     "DB_TEL"._x.PosRear;
      JNB   _007;
      L     0;
      T     "DB_TEL"._x.TargetPos;
_007: NOP   0;
      A     L 20.0;
      A     "INOUT".I_TRO.TEL_Plus;
      A(;
      O     "F_GBL_RECV".Signal31;
      ON    "DB_TEL"._x.InPosCenter;
      );
      AN    "INOUT".I_TRO.TEL_Minus;
      FP    "Tel_pFl_manPlusPos";
      =     L 20.1;
      A     L 20.1;
      JNB   _008;
      L     "DB_TargetData".Hookdata.TelPos_1.TelPos;
      T     "DB_TEL"._x.TargetPos;
_008: NOP   0;
      A     L 20.1;
      A(;
      L     "DB_TEL"._x.ActualPos;
      L     6;
      ==I;
      );
      A(;
      L     "DB_TargetData".Hookdata.TelPos_2.TelPos;
      L     0;
      <>I;
      );
      JNB   _009;
      L     "DB_TargetData".Hookdata.TelPos_2.TelPos;
      T     "DB_TEL"._x.TargetPos;
_009: NOP   0;
      A     L 20.1;
      AN    "DB_TEL"._x.InPosCenter;
      A(;
      L     "DB_TEL"._x.TargetPos;
      L     -1;
      <>I;
      );
      A     "DB_TEL"._x.PosFront;
      JNB   _00a;
      L     0;
      T     "DB_TEL"._x.TargetPos;
_00a: NOP   0;
NETWORK
TITLE = check target value
      A     "ON";
      A(;
      L     "DB_TEL"._x.TargetPos;
      L     0;
      >=I;
      );
      A(;
      L     "DB_TEL"._x.TargetPos;
      L     9;
      <=I;
      );
      =     #tmp_TargetValueOK;
NETWORK
TITLE = start motor
      A(;
      O     "DB_TEL"._x.RelForPos;
      O     "ON";
      );
      A     #tmp_TargetValueOK;
      A     "ModeAuto";
      A(;
      A     "DB_TEL"._x.TargIsPos;
      AN    "DB_TEL"._x.TargIsInternPos;
      AN    "DB_TEL"._x.TargIsCenter;
      O;
      AN    "DB_TEL"._x.TargIsPos;
      A     "DB_TEL"._x.TargIsInternPos;
      AN    "DB_TEL"._x.TargIsCenter;
      O;
      AN    "DB_TEL"._x.TargIsPos;
      AN    "DB_TEL"._x.TargIsInternPos;
      A     "DB_TEL"._x.TargIsCenter;
      );
      AN    "DB_TEL"._x.AutoInPos;
      =     "DB_TEL"._x.StartPos;
